// TIA Portal V19 program export: 0 tag tables, 0 data types, 19 data blocks, 51 code blocks (in call order from the OBs), 28 instance data blocks

DATA_BLOCK "A03_DEBUG"   // DB165
// stored: MemoryReserve 100
   VAR
      Force_Sinamics_Infeed_ON : Bool;
      Force_Sinamics_Drives_CtrlSafe : Bool;
      Forse_Contactors_CtrlSafe : Bool;
      LsStratoDepositato : Bool;
      CIn_Manager_DEBUG : Struct
         PareggiatoreTesta : Struct
            Ax : "Positioning_EPOS_Machine_COut";
         END_STRUCT;
         PareggiatoreCoda : Struct
            Ax : "Positioning_EPOS_Machine_COut";
         END_STRUCT;
         Spalle : Struct
            Testa : Struct
               Ax : "Positioning_DOL_Machine_COut";
            END_STRUCT;
            Coda : Struct
               Ax : "Positioning_DOL_Machine_COut";
            END_STRUCT;
         END_STRUCT;
         Spintore : Struct
            Vrt : "ValveMachine_COut";
            Orz : "ValveMachine_COut";
         END_STRUCT;
         TraslazioneStrato : Struct
            Ax_Testa : "Positioning_EPOS_Machine_COut";
            Ax_Coda : "Positioning_EPOS_Machine_COut";
            Manip_Sostegno : "ValveMachine_COut";
            Manip_Pareggiatore : "ValveMachine_COut";
            SostegnoVrt : "ValveMachine_COut";
         END_STRUCT;
         Sollevamento : Struct
            Ax_Testa : "Positioning_DOL_Machine_COut";
            Ax_Coda : "Positioning_DOL_Machine_COut";
         END_STRUCT;
         Sostegno : Struct
            Testa : Struct
               Ax : "Positioning_DOL_Machine_COut";
               Paletto : Struct
                  CtrlSafe : Bool;
                  Standstill : Bool;
                  Rest_CheckNext : Bool;
                  Work_CheckNext : Bool;
                  Pos : Int;
                  RestPosition : Bool;
               END_STRUCT;
            END_STRUCT;
            Coda : Struct
               Ax : "Positioning_DOL_Machine_COut";
               Paletto : Struct
                  CtrlSafe : Bool;
                  Standstill : Bool;
                  Rest_CheckNext : Bool;
                  Work_CheckNext : Bool;
                  Pos : Int;
                  RestPosition : Bool;
               END_STRUCT;
            END_STRUCT;
         END_STRUCT;
         Navetta : Struct
            ReadyToRecive : Bool;
            OutOfWorkspace : Bool;
            InPosizioneDiDeposito : Bool;
            RequestDeposito : Bool;
         END_STRUCT;
         RegolazBord : Struct
            CassettaOP : Real := 65.0;
            LineSetupExe : Bool;
         END_STRUCT;
      END_STRUCT;
      CIn_Manager04_Debug : Struct
         Navetta : Struct
            Testa : Struct
               Ax : "Positioning_DOL_Machine_COut";
               PalettiEsterni : "ValveMachine_COut";
               PalettiInterni : "ValveMachine_COut";
            END_STRUCT;
            Coda : Struct
               Ax : "Positioning_DOL_Machine_COut";
               PalettiEsterni : "ValveMachine_COut";
               PalettiInterni : "ValveMachine_COut";
            END_STRUCT;
            Cumulativo : Struct
               PalettiEsterni : "ValveMachine_COut";
               PalettiInterni : "ValveMachine_COut";
            END_STRUCT;
         END_STRUCT;
         Sollevamento : Struct
            ReadyToDrop : Bool;   // In posizione di deposito e pacco completato
         END_STRUCT;
         Antiribaltamento : Struct
            Work : Bool;
            Rest : Bool;
         END_STRUCT;
      END_STRUCT;
   END_VAR
   VAR RETAIN
      HU_Test : Struct
         Enable : Bool;
         EnableDrive : Bool;
         "Req_Par-Bloccaggio" : Bool;
         "Req_Par-Paregg" : Bool;
         Ctrl_Safe : Bool;
      END_STRUCT;
   END_VAR
   VAR
      test_bitA : Bool;
      test_bitB : Bool;
   END_VAR
   VAR RETAIN
      A0301_Manager : Struct
         BeamCode : Bool;   // 0=Solo Part / 1 = Accoppiamento Part
         "Case" : Int;
         "P1-P3_Init" : Bool;
         "P1-P2_Init" : Bool;
         TrasportoStart : Bool;
         PTrk_Pos1_Write : Bool;
      END_STRUCT;
      A0302_Manager : Struct
         BeamCode : Bool;   // 0=Solo Part / 1 = Accoppiamento Part
         JMP : Bool := TRUE;
         A0303_ReadyToRecive : Bool;
         PareggiaRead : Bool;
         AttrezzamentoBordatrice : Bool;
         BTrk_EXIT_Clear : Bool;
      END_STRUCT;
   END_VAR
   VAR
      A301_PTrk : "PTrk_Item";
   END_VAR
BEGIN
   A301_PTrk.O_ID := 1;
   A301_PTrk.C_ID := 0;
   A301_PTrk.Quality := 0;
   A301_PTrk.Beam_Code := 1;
   A301_PTrk.PLen_Meas := 2700.0;
   A301_PTrk.W_A := 140.0;
   A301_PTrk.H_B := 4.5;
   A301_PTrk.ShiftDone := FALSE;
END_DATA_BLOCK

DATA_BLOCK "PrjConfig_A03"   // DB82
// stored: MemoryReserve 100
   VAR
      Area03_Main : "AreaConfig";
   END_VAR
   VAR RETAIN
      A0301 : Struct
         Fermi_P1 : Struct
            Fermi : Array[1..6] of "ValveMachine_Config";
            Sfalsatore : "ValveMachine_Config";
            DelayMissingCondition : Time := T#3S;
         END_STRUCT;
         Fermi_P2 : Struct
            Fermi : Array[1..6] of "ValveMachine_Config";
            Sollevatori : Array[1..6] of "ValveMachine_Config";
            DelayMissingCondition : Time := T#3S;
         END_STRUCT;
         Fermi_P3 : Struct
            Fermi : Array[1..6] of "ValveMachine_Config";
            DelayMissingCondition : Time := T#3S;
         END_STRUCT;
         Fermi_P4 : Struct
            Fermi : Array[1..6] of "ValveMachine_Config";
            DelayMissingCondition : Time := T#3S;
         END_STRUCT;
         Trasporto { S7_SetPoint := 'True'} : "SpeedMachine_Config";
         Ribaltatore : Struct
            Ax : "Positioning_EPOS_Machine_Config_NEW";
            Solleva_Rib : Array[1..6] of "ValveMachine_Config";
         END_STRUCT;
         SpintoreLaterale : Struct
            Vrt_1 : "ValveMachine_Config";
            Orz_1 : "ValveMachine_Config";
            Vrt_2 : "ValveMachine_Config";
            Orz_2 : "ValveMachine_Config";
            Sollevatori : Array[1..7] of "ValveMachine_Config";
            QuotaIngombro_SpinLat2 : Real := 2680.0;
            QuotaIngombro_SpinLat1 { ExternalWritable := 'False'} : Real := 4777.0;
            DelayMissingCondition : Time := T#500MS;
         END_STRUCT;
      END_STRUCT;
      A0302 : Struct
         Spintore : Struct
            Ax : "Positioning_EPOS_Machine_Config_NEW";
            Vrt : "ValveMachine_Config";
            Orz : "ValveMachine_Config";
            SpintoreLat : Struct
               QuotaIngombro_SpinLat2 : Real := 2680.0;
               QuotaIngombro_SpinLat1 : Real := 4777.0;
            END_STRUCT;
            Bordatrice : Struct
               QuotaIngresso : Real := 801.0;
            END_STRUCT;
            DelayMissingCondition : Time := T#0MS;
         END_STRUCT;
         Bordatrice : Struct
            Ax : "Positioning_EPOS_Machine_Config_NEW";
            Measure : Struct
               K1_CarroPost : LReal := 674.0;   // K1: Misura tra carro di coda e sensore applicato per controllo ingombro pezzo con carro giù
               K2_BancoIngresso : LReal := 3560.0;   // K2: Misura interasse tra lo 0 al centro del banco e la FTC all'uscita della Bordatrice
            END_STRUCT;
         END_STRUCT;
         Regolaz_Bordatrice : Struct
            Formato : Struct
               Ax_D : Array[1..1] of "Positioning_DOL_Machine_Config";
               Ax_M : Array[1..10] of "Positioning_MOL_Machine_Config";
               M1_1 : "Positioning_DOL_Machine_Config";
               M1_2 : "Positioning_DOL_Machine_Config";
               M1_3 : "Positioning_MOL_Machine_Config";
               M1_4 : "Positioning_MOL_Machine_Config";
            END_STRUCT;
         END_STRUCT;
         Rulliera : Struct
            Ax : "SpeedMachine_Config";
         END_STRUCT;
         Centratori : Struct
            Centraggio : Array[1..3] of "ValveMachine_Config";
            Sollevamento : Array[1..3] of "ValveMachine_Config";
            DelayMissingCondition : Time := T#500MS;
            WorkWindows : Struct   // Finestre di disattivazione Centratore 1 e 3 in funzione dei Carri
               Coda : Struct
                  Min : LReal := 300.0;
                  Max : LReal := 1378.0;
               END_STRUCT;
               Testa : Struct
                  Min : LReal := 433.0;
                  Max : LReal := 970.0;
               END_STRUCT;
            END_STRUCT;
         END_STRUCT;
         PareggiatoreCoda : Struct
            Ax : "Positioning_DOL_Machine_Config";
            Bloccaggio : "ValveMachine_Config";
            BattutaVerticale : "ValveMachine_Config";
            PareggiatoreLong : "ValveMachine_Config";
            PosPareggiatore : Struct
               QuotaMin_Work : LReal := 82.0;
               QuotaMax_Work { S7_SetPoint := 'True'} : LReal := 91.0;
            END_STRUCT;
            MinDistanzaConSpalla { S7_SetPoint := 'True'} : LReal := 85.7;
            DelayMissingCondition : Time := T#200MS;
         END_STRUCT;
         PareggiatoreTesta : Struct
            Ax : "Positioning_DOL_Machine_Config";
            Bloccaggio : "ValveMachine_Config";
            Sollevamento : "ValveMachine_Config";
            Centraggio : "ValveMachine_Config";
            MinDistanzaConSpalla : LReal := 5.0;
            DelayMissingCondition : Time := T#200MS;
         END_STRUCT;
         Manipolatore : Struct
            Testa : Struct
               Ax : "Positioning_EPOS_Machine_Config_NEW";
               Sollevatore : "ValveMachine_Config";
               Magnete : "ValveMachine_Config";
            END_STRUCT;
            Coda : Struct
               Ax : "Positioning_EPOS_Machine_Config_NEW";
               Sollevatore : "ValveMachine_Config";
               Magnete : "ValveMachine_Config";
            END_STRUCT;
            DelayMissingCondition : Time := T#200MS;
         END_STRUCT;
      END_STRUCT;
   END_VAR
BEGIN
   Area03_Main.TimeOutStopImmediate := T#1S_500MS;
   Area03_Main.TimeOutStopInPhase := T#10S;
   Area03_Main.TimeOutStopProgrammed := T#5M;
   Area03_Main.TimeOutResetAlarms := T#1S;
   A0301.Fermi_P1.Fermi[1..6].DelayPressureRunningTimeout := T#3S;
   A0301.Fermi_P1.Fermi[1..6].DelayMissingCondition := T#3S;
   A0301.Fermi_P1.Fermi[1..6].Rest_LsQty := 1;
   A0301.Fermi_P1.Fermi[1..6].Work_LsQty := 0;
   A0301.Fermi_P1.Fermi[1..6].Rest_RetainAut := FALSE;
   A0301.Fermi_P1.Fermi[1..6].Work_RetainAut := FALSE;
   A0301.Fermi_P1.Fermi[1..6].V.RestLimSwitchExist := TRUE;
   A0301.Fermi_P1.Fermi[1..6].V.WorkLimSwitchExist := FALSE;
   A0301.Fermi_P1.Fermi[1..6].V.CheckOilInPressure := FALSE;
   A0301.Fermi_P1.Fermi[1..6].V.CutRestWhenIsAtRest := TRUE;
   A0301.Fermi_P1.Fermi[1..6].V.CutWorkWhenIsAtWork := FALSE;
   A0301.Fermi_P1.Fermi[1..6].V.RestTime := T#1MS;
   A0301.Fermi_P1.Fermi[1..6].V.WorkTime := T#100MS;
   A0301.Fermi_P1.Fermi[1..6].V.RestTimeOut := T#4S;
   A0301.Fermi_P1.Fermi[1..6].V.WorkTimeOut := T#4S;
   A0301.Fermi_P1.Sfalsatore.DelayPressureRunningTimeout := T#3S;
   A0301.Fermi_P1.Sfalsatore.DelayMissingCondition := T#3S;
   A0301.Fermi_P1.Sfalsatore.Rest_LsQty := 1;
   A0301.Fermi_P1.Sfalsatore.Work_LsQty := 1;
   A0301.Fermi_P1.Sfalsatore.Rest_RetainAut := FALSE;
   A0301.Fermi_P1.Sfalsatore.Work_RetainAut := FALSE;
   A0301.Fermi_P1.Sfalsatore.V.RestLimSwitchExist := TRUE;
   A0301.Fermi_P1.Sfalsatore.V.WorkLimSwitchExist := TRUE;
   A0301.Fermi_P1.Sfalsatore.V.CheckOilInPressure := FALSE;
   A0301.Fermi_P1.Sfalsatore.V.CutRestWhenIsAtRest := FALSE;
   A0301.Fermi_P1.Sfalsatore.V.CutWorkWhenIsAtWork := TRUE;
   A0301.Fermi_P1.Sfalsatore.V.RestTime := T#1S;
   A0301.Fermi_P1.Sfalsatore.V.WorkTime := T#300MS;
   A0301.Fermi_P1.Sfalsatore.V.RestTimeOut := T#1H;
   A0301.Fermi_P1.Sfalsatore.V.WorkTimeOut := T#1H;
   A0301.Fermi_P2.Fermi[1..6].DelayPressureRunningTimeout := T#3S;
   A0301.Fermi_P2.Fermi[1..6].DelayMissingCondition := T#3S;
   A0301.Fermi_P2.Fermi[1..6].Rest_LsQty := 1;
   A0301.Fermi_P2.Fermi[1..6].Work_LsQty := 0;
   A0301.Fermi_P2.Fermi[1..6].Rest_RetainAut := FALSE;
   A0301.Fermi_P2.Fermi[1..6].Work_RetainAut := FALSE;
   A0301.Fermi_P2.Fermi[1..6].V.RestLimSwitchExist := TRUE;
   A0301.Fermi_P2.Fermi[1..6].V.WorkLimSwitchExist := FALSE;
   A0301.Fermi_P2.Fermi[1..6].V.CheckOilInPressure := FALSE;
   A0301.Fermi_P2.Fermi[1..6].V.CutRestWhenIsAtRest := TRUE;
   A0301.Fermi_P2.Fermi[1..6].V.CutWorkWhenIsAtWork := FALSE;
   A0301.Fermi_P2.Fermi[1..6].V.RestTime := T#1MS;
   A0301.Fermi_P2.Fermi[1..6].V.WorkTime := T#100MS;
   A0301.Fermi_P2.Fermi[1..6].V.RestTimeOut := T#4S;
   A0301.Fermi_P2.Fermi[1..6].V.WorkTimeOut := T#4S;
   A0301.Fermi_P2.Sollevatori[1..6].DelayPressureRunningTimeout := T#3S;
   A0301.Fermi_P2.Sollevatori[1..6].DelayMissingCondition := T#3S;
   A0301.Fermi_P2.Sollevatori[1..6].Rest_LsQty := 1;
   A0301.Fermi_P2.Sollevatori[1..6].Work_LsQty := 0;
   A0301.Fermi_P2.Sollevatori[1..6].Rest_RetainAut := FALSE;
   A0301.Fermi_P2.Sollevatori[1..6].Work_RetainAut := FALSE;
   A0301.Fermi_P2.Sollevatori[1..6].V.RestLimSwitchExist := TRUE;
   A0301.Fermi_P2.Sollevatori[1..6].V.WorkLimSwitchExist := FALSE;
   A0301.Fermi_P2.Sollevatori[1..6].V.CheckOilInPressure := FALSE;
   A0301.Fermi_P2.Sollevatori[1..6].V.CutRestWhenIsAtRest := TRUE;
   A0301.Fermi_P2.Sollevatori[1..6].V.CutWorkWhenIsAtWork := FALSE;
   A0301.Fermi_P2.Sollevatori[1..6].V.RestTime := T#1MS;
   A0301.Fermi_P2.Sollevatori[1..6].V.WorkTime := T#100MS;
   A0301.Fermi_P2.Sollevatori[1..6].V.RestTimeOut := T#4S;
   A0301.Fermi_P2.Sollevatori[1..6].V.WorkTimeOut := T#4S;
   A0301.Fermi_P3.Fermi[1..6].DelayPressureRunningTimeout := T#3S;
   A0301.Fermi_P3.Fermi[1..6].DelayMissingCondition := T#3S;
   A0301.Fermi_P3.Fermi[1..6].Rest_LsQty := 1;
   A0301.Fermi_P3.Fermi[1..6].Work_LsQty := 0;
   A0301.Fermi_P3.Fermi[1..6].Rest_RetainAut := FALSE;
   A0301.Fermi_P3.Fermi[1..6].Work_RetainAut := FALSE;
   A0301.Fermi_P3.Fermi[1..6].V.RestLimSwitchExist := TRUE;
   A0301.Fermi_P3.Fermi[1..6].V.WorkLimSwitchExist := FALSE;
   A0301.Fermi_P3.Fermi[1..6].V.CheckOilInPressure := FALSE;
   A0301.Fermi_P3.Fermi[1..6].V.CutRestWhenIsAtRest := TRUE;
   A0301.Fermi_P3.Fermi[1..6].V.CutWorkWhenIsAtWork := FALSE;
   A0301.Fermi_P3.Fermi[1..6].V.RestTime := T#1MS;
   A0301.Fermi_P3.Fermi[1..6].V.WorkTime := T#100MS;
   A0301.Fermi_P3.Fermi[1..6].V.RestTimeOut := T#4S;
   A0301.Fermi_P3.Fermi[1..6].V.WorkTimeOut := T#4S;
   A0301.Fermi_P4.Fermi[1..6].DelayPressureRunningTimeout := T#3S;
   A0301.Fermi_P4.Fermi[1..6].DelayMissingCondition := T#3S;
   A0301.Fermi_P4.Fermi[1..6].Rest_LsQty := 1;
   A0301.Fermi_P4.Fermi[1..6].Work_LsQty := 0;
   A0301.Fermi_P4.Fermi[1..6].Rest_RetainAut := FALSE;
   A0301.Fermi_P4.Fermi[1..6].Work_RetainAut := FALSE;
   A0301.Fermi_P4.Fermi[1..6].V.RestLimSwitchExist := TRUE;
   A0301.Fermi_P4.Fermi[1..6].V.WorkLimSwitchExist := FALSE;
   A0301.Fermi_P4.Fermi[1..6].V.CheckOilInPressure := FALSE;
   A0301.Fermi_P4.Fermi[1..6].V.CutRestWhenIsAtRest := TRUE;
   A0301.Fermi_P4.Fermi[1..6].V.CutWorkWhenIsAtWork := FALSE;
   A0301.Fermi_P4.Fermi[1..6].V.RestTime := T#1MS;
   A0301.Fermi_P4.Fermi[1..6].V.WorkTime := T#300MS;
   A0301.Fermi_P4.Fermi[1..6].V.RestTimeOut := T#4S;
   A0301.Fermi_P4.Fermi[1..6].V.WorkTimeOut := T#4S;
   A0301.Trasporto.SLS_VEL := 5000.0;
   A0301.Trasporto.DelayMissingCondition := T#3S;
   A0301.Trasporto.Ax.SINA_Drive.ReferenceVelocity := 2200.0;
   A0301.Trasporto.Ax.SINA_Drive.InvertDirection := FALSE;
   A0301.Trasporto.Ax.MinAccTime := 0.1;
   A0301.Trasporto.Ax.MinDecTime := 0.1;
   A0301.Trasporto.Ax.LeadScrewPitchVal := 359.8;
   A0301.Trasporto.Ax.MotorRevolution := 20.0;
   A0301.Trasporto.Ax.LoadRevolution := 1.0;
   A0301.Trasporto.Ax.PowerOffDelay := T#1S_500MS;
   A0301.Trasporto.Ax.StandstillVelocity := 50.0;
   A0301.Trasporto.Ax.StandstillDelay := T#100MS;
   A0301.Trasporto.Fan.Presence := FALSE;
   A0301.Trasporto.Fan.DelayOff := T#0MS;
   A0301.Trasporto.Brake_Presence := FALSE;
   A0301.Ribaltatore.Ax.SLS_Vel := 3000.0;
   A0301.Ribaltatore.Ax.DelayMissingCondition := T#100MS;
   A0301.Ribaltatore.Ax.Ax.Encoder_Inc_AutoReloadPosition := FALSE;
   A0301.Ribaltatore.Ax.Ax.Encoder_is_Absolute := TRUE;
   A0301.Ribaltatore.Ax.Ax.LeadScrewPitchVal := 9.0000015;
   A0301.Ribaltatore.Ax.Ax.MotorRevolution := 23.33;
   A0301.Ribaltatore.Ax.Ax.LoadRevolution := 1.0;
   A0301.Ribaltatore.Ax.Ax.PowerOffDelay := T#100MS;
   A0301.Ribaltatore.Ax.Ax.MaxRPM_S120_P2000 := 3000.0;
   A0301.Ribaltatore.Ax.Ax.MaxVel_S120_P2571 := 6000.0;
   A0301.Ribaltatore.Ax.Ax.MaxAcc_S120_P2572 := 50.0;
   A0301.Ribaltatore.Ax.Ax.MaxDec_S120_P2573 := 50.0;
   A0301.Ribaltatore.Ax.Ax.Modulo_S120_P2566 := 0.0;
   A0301.Ribaltatore.Ax.Ax.SwLimMinus_S120_P2580 := 0.25;
   A0301.Ribaltatore.Ax.Ax.SwLimPlus_S120_P2581 := 125.0;
   A0301.Ribaltatore.Ax.Fan.Presence := FALSE;
   A0301.Ribaltatore.Ax.Fan.DelayOff := T#0MS;
   A0301.Ribaltatore.Ax.Brake_Presence := FALSE;
   A0301.Ribaltatore.Solleva_Rib[1..6].DelayPressureRunningTimeout := T#3S;
   A0301.Ribaltatore.Solleva_Rib[1..6].DelayMissingCondition := T#3S;
   A0301.Ribaltatore.Solleva_Rib[1..6].Rest_LsQty := 1;
   A0301.Ribaltatore.Solleva_Rib[1..6].Work_LsQty := 1;
   A0301.Ribaltatore.Solleva_Rib[1..6].Rest_RetainAut := FALSE;
   A0301.Ribaltatore.Solleva_Rib[1..6].Work_RetainAut := FALSE;
   A0301.Ribaltatore.Solleva_Rib[1..6].V.RestLimSwitchExist := TRUE;
   A0301.Ribaltatore.Solleva_Rib[1..6].V.WorkLimSwitchExist := TRUE;
   A0301.Ribaltatore.Solleva_Rib[1..6].V.CheckOilInPressure := FALSE;
   A0301.Ribaltatore.Solleva_Rib[1..6].V.CutRestWhenIsAtRest := FALSE;
   A0301.Ribaltatore.Solleva_Rib[1..6].V.CutWorkWhenIsAtWork := FALSE;
   A0301.Ribaltatore.Solleva_Rib[1..6].V.RestTime := T#1MS;
   A0301.Ribaltatore.Solleva_Rib[1..6].V.WorkTime := T#200MS;
   A0301.Ribaltatore.Solleva_Rib[1..6].V.RestTimeOut := T#5S;
   A0301.Ribaltatore.Solleva_Rib[1..6].V.WorkTimeOut := T#5S;
   A0301.SpintoreLaterale.Vrt_1.DelayPressureRunningTimeout := T#3S;
   A0301.SpintoreLaterale.Vrt_1.DelayMissingCondition := T#3S;
   A0301.SpintoreLaterale.Vrt_1.Rest_LsQty := 1;
   A0301.SpintoreLaterale.Vrt_1.Work_LsQty := 0;
   A0301.SpintoreLaterale.Vrt_1.Rest_RetainAut := FALSE;
   A0301.SpintoreLaterale.Vrt_1.Work_RetainAut := FALSE;
   A0301.SpintoreLaterale.Vrt_1.V.RestLimSwitchExist := TRUE;
   A0301.SpintoreLaterale.Vrt_1.V.WorkLimSwitchExist := FALSE;
   A0301.SpintoreLaterale.Vrt_1.V.CheckOilInPressure := FALSE;
   A0301.SpintoreLaterale.Vrt_1.V.CutRestWhenIsAtRest := TRUE;
   A0301.SpintoreLaterale.Vrt_1.V.CutWorkWhenIsAtWork := FALSE;
   A0301.SpintoreLaterale.Vrt_1.V.RestTime := T#1MS;
   A0301.SpintoreLaterale.Vrt_1.V.WorkTime := T#300MS;
   A0301.SpintoreLaterale.Vrt_1.V.RestTimeOut := T#5S;
   A0301.SpintoreLaterale.Vrt_1.V.WorkTimeOut := T#5S;
   A0301.SpintoreLaterale.Orz_1.DelayPressureRunningTimeout := T#3S;
   A0301.SpintoreLaterale.Orz_1.DelayMissingCondition := T#3S;
   A0301.SpintoreLaterale.Orz_1.Rest_LsQty := 1;
   A0301.SpintoreLaterale.Orz_1.Work_LsQty := 0;
   A0301.SpintoreLaterale.Orz_1.Rest_RetainAut := FALSE;
   A0301.SpintoreLaterale.Orz_1.Work_RetainAut := FALSE;
   A0301.SpintoreLaterale.Orz_1.V.RestLimSwitchExist := TRUE;
   A0301.SpintoreLaterale.Orz_1.V.WorkLimSwitchExist := FALSE;
   A0301.SpintoreLaterale.Orz_1.V.CheckOilInPressure := FALSE;
   A0301.SpintoreLaterale.Orz_1.V.CutRestWhenIsAtRest := FALSE;
   A0301.SpintoreLaterale.Orz_1.V.CutWorkWhenIsAtWork := FALSE;
   A0301.SpintoreLaterale.Orz_1.V.RestTime := T#1MS;
   A0301.SpintoreLaterale.Orz_1.V.WorkTime := T#300MS;
   A0301.SpintoreLaterale.Orz_1.V.RestTimeOut := T#5S;
   A0301.SpintoreLaterale.Orz_1.V.WorkTimeOut := T#5S;
   A0301.SpintoreLaterale.Vrt_2.DelayPressureRunningTimeout := T#3S;
   A0301.SpintoreLaterale.Vrt_2.DelayMissingCondition := T#3S;
   A0301.SpintoreLaterale.Vrt_2.Rest_LsQty := 1;
   A0301.SpintoreLaterale.Vrt_2.Work_LsQty := 0;
   A0301.SpintoreLaterale.Vrt_2.Rest_RetainAut := FALSE;
   A0301.SpintoreLaterale.Vrt_2.Work_RetainAut := FALSE;
   A0301.SpintoreLaterale.Vrt_2.V.RestLimSwitchExist := TRUE;
   A0301.SpintoreLaterale.Vrt_2.V.WorkLimSwitchExist := FALSE;
   A0301.SpintoreLaterale.Vrt_2.V.CheckOilInPressure := FALSE;
   A0301.SpintoreLaterale.Vrt_2.V.CutRestWhenIsAtRest := TRUE;
   A0301.SpintoreLaterale.Vrt_2.V.CutWorkWhenIsAtWork := FALSE;
   A0301.SpintoreLaterale.Vrt_2.V.RestTime := T#1MS;
   A0301.SpintoreLaterale.Vrt_2.V.WorkTime := T#300MS;
   A0301.SpintoreLaterale.Vrt_2.V.RestTimeOut := T#5S;
   A0301.SpintoreLaterale.Vrt_2.V.WorkTimeOut := T#5S;
   A0301.SpintoreLaterale.Orz_2.DelayPressureRunningTimeout := T#3S;
   A0301.SpintoreLaterale.Orz_2.DelayMissingCondition := T#3S;
   A0301.SpintoreLaterale.Orz_2.Rest_LsQty := 1;
   A0301.SpintoreLaterale.Orz_2.Work_LsQty := 0;
   A0301.SpintoreLaterale.Orz_2.Rest_RetainAut := FALSE;
   A0301.SpintoreLaterale.Orz_2.Work_RetainAut := FALSE;
   A0301.SpintoreLaterale.Orz_2.V.RestLimSwitchExist := TRUE;
   A0301.SpintoreLaterale.Orz_2.V.WorkLimSwitchExist := FALSE;
   A0301.SpintoreLaterale.Orz_2.V.CheckOilInPressure := FALSE;
   A0301.SpintoreLaterale.Orz_2.V.CutRestWhenIsAtRest := FALSE;
   A0301.SpintoreLaterale.Orz_2.V.CutWorkWhenIsAtWork := FALSE;
   A0301.SpintoreLaterale.Orz_2.V.RestTime := T#1MS;
   A0301.SpintoreLaterale.Orz_2.V.WorkTime := T#300MS;
   A0301.SpintoreLaterale.Orz_2.V.RestTimeOut := T#5S;
   A0301.SpintoreLaterale.Orz_2.V.WorkTimeOut := T#5S;
   A0301.SpintoreLaterale.Sollevatori[1..7].DelayPressureRunningTimeout := T#3S;
   A0301.SpintoreLaterale.Sollevatori[1..7].DelayMissingCondition := T#3S;
   A0301.SpintoreLaterale.Sollevatori[1..7].Rest_LsQty := 1;
   A0301.SpintoreLaterale.Sollevatori[1..7].Work_LsQty := 0;
   A0301.SpintoreLaterale.Sollevatori[1..7].Rest_RetainAut := FALSE;
   A0301.SpintoreLaterale.Sollevatori[1..7].Work_RetainAut := FALSE;
   A0301.SpintoreLaterale.Sollevatori[1..7].V.RestLimSwitchExist := TRUE;
   A0301.SpintoreLaterale.Sollevatori[1..7].V.WorkLimSwitchExist := FALSE;
   A0301.SpintoreLaterale.Sollevatori[1..7].V.CheckOilInPressure := FALSE;
   A0301.SpintoreLaterale.Sollevatori[1..7].V.CutRestWhenIsAtRest := TRUE;
   A0301.SpintoreLaterale.Sollevatori[1..7].V.CutWorkWhenIsAtWork := TRUE;
   A0301.SpintoreLaterale.Sollevatori[1..7].V.RestTime := T#1S;
   A0301.SpintoreLaterale.Sollevatori[1..7].V.WorkTime := T#500MS;
   A0301.SpintoreLaterale.Sollevatori[1..7].V.RestTimeOut := T#4S;
   A0301.SpintoreLaterale.Sollevatori[1..7].V.WorkTimeOut := T#4S;
   A0302.Spintore.Ax.SLS_Vel := 3000.0;
   A0302.Spintore.Ax.DelayMissingCondition := T#1S;
   A0302.Spintore.Ax.Ax.Encoder_Inc_AutoReloadPosition := FALSE;
   A0302.Spintore.Ax.Ax.Encoder_is_Absolute := TRUE;
   A0302.Spintore.Ax.Ax.LeadScrewPitchVal := 287.989799;
   A0302.Spintore.Ax.Ax.MotorRevolution := 10.0;
   A0302.Spintore.Ax.Ax.LoadRevolution := 1.0;
   A0302.Spintore.Ax.Ax.PowerOffDelay := T#1S;
   A0302.Spintore.Ax.Ax.MaxRPM_S120_P2000 := 3000.0;
   A0302.Spintore.Ax.Ax.MaxVel_S120_P2571 := 86396.0;
   A0302.Spintore.Ax.Ax.MaxAcc_S120_P2572 := 5000.0;
   A0302.Spintore.Ax.Ax.MaxDec_S120_P2573 := 5000.0;
   A0302.Spintore.Ax.Ax.Modulo_S120_P2566 := 0.0;
   A0302.Spintore.Ax.Ax.SwLimMinus_S120_P2580 := 0.5;
   A0302.Spintore.Ax.Ax.SwLimPlus_S120_P2581 := 5370.0;
   A0302.Spintore.Ax.Fan.Presence := FALSE;
   A0302.Spintore.Ax.Fan.DelayOff := T#0MS;
   A0302.Spintore.Ax.Brake_Presence := FALSE;
   A0302.Spintore.Vrt.DelayPressureRunningTimeout := T#3S;
   A0302.Spintore.Vrt.DelayMissingCondition := T#3S;
   A0302.Spintore.Vrt.Rest_LsQty := 1;
   A0302.Spintore.Vrt.Work_LsQty := 1;
   A0302.Spintore.Vrt.Rest_RetainAut := FALSE;
   A0302.Spintore.Vrt.Work_RetainAut := FALSE;
   A0302.Spintore.Vrt.V.RestLimSwitchExist := TRUE;
   A0302.Spintore.Vrt.V.WorkLimSwitchExist := TRUE;
   A0302.Spintore.Vrt.V.CheckOilInPressure := FALSE;
   A0302.Spintore.Vrt.V.CutRestWhenIsAtRest := TRUE;
   A0302.Spintore.Vrt.V.CutWorkWhenIsAtWork := FALSE;
   A0302.Spintore.Vrt.V.RestTime := T#10MS;
   A0302.Spintore.Vrt.V.WorkTime := T#100MS;
   A0302.Spintore.Vrt.V.RestTimeOut := T#4S;
   A0302.Spintore.Vrt.V.WorkTimeOut := T#4S;
   A0302.Spintore.Orz.DelayPressureRunningTimeout := T#3S;
   A0302.Spintore.Orz.DelayMissingCondition := T#3S;
   A0302.Spintore.Orz.Rest_LsQty := 1;
   A0302.Spintore.Orz.Work_LsQty := 0;
   A0302.Spintore.Orz.Rest_RetainAut := FALSE;
   A0302.Spintore.Orz.Work_RetainAut := FALSE;
   A0302.Spintore.Orz.V.RestLimSwitchExist := TRUE;
   A0302.Spintore.Orz.V.WorkLimSwitchExist := FALSE;
   A0302.Spintore.Orz.V.CheckOilInPressure := FALSE;
   A0302.Spintore.Orz.V.CutRestWhenIsAtRest := TRUE;
   A0302.Spintore.Orz.V.CutWorkWhenIsAtWork := FALSE;
   A0302.Spintore.Orz.V.RestTime := T#10MS;
   A0302.Spintore.Orz.V.WorkTime := T#100MS;
   A0302.Spintore.Orz.V.RestTimeOut := T#4S;
   A0302.Spintore.Orz.V.WorkTimeOut := T#4S;
   A0302.Bordatrice.Ax.SLS_Vel := 3000.0;
   A0302.Bordatrice.Ax.DelayMissingCondition := T#200MS;
   A0302.Bordatrice.Ax.Ax.Encoder_Inc_AutoReloadPosition := TRUE;
   A0302.Bordatrice.Ax.Ax.Encoder_is_Absolute := FALSE;
   A0302.Bordatrice.Ax.Ax.LeadScrewPitchVal := 486.946;
   A0302.Bordatrice.Ax.Ax.MotorRevolution := 12.4;
   A0302.Bordatrice.Ax.Ax.LoadRevolution := 1.0;
   A0302.Bordatrice.Ax.Ax.PowerOffDelay := T#500MS;
   A0302.Bordatrice.Ax.Ax.MaxRPM_S120_P2000 := 3000.0;
   A0302.Bordatrice.Ax.Ax.MaxVel_S120_P2571 := 60000.0;
   A0302.Bordatrice.Ax.Ax.MaxAcc_S120_P2572 := 4000.0;
   A0302.Bordatrice.Ax.Ax.MaxDec_S120_P2573 := 4000.0;
   A0302.Bordatrice.Ax.Ax.Modulo_S120_P2566 := 1000000000.0;
   A0302.Bordatrice.Ax.Ax.SwLimMinus_S120_P2580 := 0.0;
   A0302.Bordatrice.Ax.Ax.SwLimPlus_S120_P2581 := 0.0;
   A0302.Bordatrice.Ax.Fan.Presence := FALSE;
   A0302.Bordatrice.Ax.Fan.DelayOff := T#0MS;
   A0302.Bordatrice.Ax.Brake_Presence := FALSE;
   A0302.Regolaz_Bordatrice.Formato.Ax_D[1].DelayMissingCondition := T#3S;
   A0302.Regolaz_Bordatrice.Formato.Ax_D[1].CyclicOBTime_ms := 10.0;
   A0302.Regolaz_Bordatrice.Formato.Ax_D[1].Ax.limitMinus := 59.0;
   A0302.Regolaz_Bordatrice.Formato.Ax_D[1].Ax.limitPlus := 215.0;
   A0302.Regolaz_Bordatrice.Formato.Ax_D[1].Ax.Backlash := 0.4;
   A0302.Regolaz_Bordatrice.Formato.Ax_D[1].Ax.BacklashActivation := TRUE;
   A0302.Regolaz_Bordatrice.Formato.Ax_D[1].Ax.ToleranceWindow := 0.0;
   A0302.Regolaz_Bordatrice.Formato.Ax_D[1].Ax.ToleranceWindowDelay := T#100MS;
   A0302.Regolaz_Bordatrice.Formato.Ax_D[1].Ax.PreCutOff := 0.03;
   A0302.Regolaz_Bordatrice.Formato.Ax_D[1].Ax.PreEndLowSpeed := 0.0;
   A0302.Regolaz_Bordatrice.Formato.Ax_D[1].Ax.PreEndMedSpeed := 0.0;
   A0302.Regolaz_Bordatrice.Formato.Ax_D[1].Ax.ChangeDirectionDelay := T#0MS;
   A0302.Regolaz_Bordatrice.Formato.Ax_D[1].Ax.StandstillVelocity := 0.5;
   A0302.Regolaz_Bordatrice.Formato.Ax_D[1].Ax.StandStillDelay := T#100MS;
   A0302.Regolaz_Bordatrice.Formato.Ax_D[1].Ax.HomingDirection := FALSE;
   A0302.Regolaz_Bordatrice.Formato.Ax_D[1].Ax.RecallTime := 0.0;
   A0302.Regolaz_Bordatrice.Formato.Ax_D[1].Ax.VelocityFilter_T := 10.0;
   A0302.Regolaz_Bordatrice.Formato.Ax_D[1].Ax.VelocityMeasUnit := 2;
   A0302.Regolaz_Bordatrice.Formato.Ax_D[1].Ax.PosFbkDisabled := FALSE;
   A0302.Regolaz_Bordatrice.Formato.Ax_D[1].Ax.FbkCtrlDisabled := TRUE;
   A0302.Regolaz_Bordatrice.Formato.Ax_D[1].Ax_UM2."m" := -1.0;
   A0302.Regolaz_Bordatrice.Formato.Ax_D[1].Ax_UM2.q := 320.5;
   A0302.Regolaz_Bordatrice.Formato.Ax_D[1].S120.SpeedMotor.ReferenceVelocity := 2200.0;
   A0302.Regolaz_Bordatrice.Formato.Ax_D[1].S120.SpeedMotor.InvertDirection := FALSE;
   A0302.Regolaz_Bordatrice.Formato.Ax_D[1].S120.PowerOffDelay := T#1S_500MS;
   A0302.Regolaz_Bordatrice.Formato.Ax_D[1].S120.StandstillVelocity := 20.0;
   A0302.Regolaz_Bordatrice.Formato.Ax_D[1].S120.AccTime := 0.5;
   A0302.Regolaz_Bordatrice.Formato.Ax_D[1].S120.DecTime := 0.5;
   A0302.Regolaz_Bordatrice.Formato.Ax_D[1].Fan.Presence := FALSE;
   A0302.Regolaz_Bordatrice.Formato.Ax_D[1].Fan.DelayOff := T#10M;
   A0302.Regolaz_Bordatrice.Formato.Ax_D[1].Brake_Presence := FALSE;
   A0302.Regolaz_Bordatrice.Formato.Ax_M[1..10].DelayMissingCondition := T#100MS;
   A0302.Regolaz_Bordatrice.Formato.Ax_M[1..10].CyclicOBTime_ms := 10.0;
   A0302.Regolaz_Bordatrice.Formato.Ax_M[1..10].Ax.limitMinus := 38.0;
   A0302.Regolaz_Bordatrice.Formato.Ax_M[1..10].Ax.limitPlus := 52.0;
   A0302.Regolaz_Bordatrice.Formato.Ax_M[1..10].Ax.Backlash := 0.4;
   A0302.Regolaz_Bordatrice.Formato.Ax_M[1..10].Ax.BacklashActivation := TRUE;
   A0302.Regolaz_Bordatrice.Formato.Ax_M[1..10].Ax.ToleranceWindow := 0.0;
   A0302.Regolaz_Bordatrice.Formato.Ax_M[1..10].Ax.ToleranceWindowDelay := T#100MS;
   A0302.Regolaz_Bordatrice.Formato.Ax_M[1..10].Ax.PreCutOff := 0.03;
   A0302.Regolaz_Bordatrice.Formato.Ax_M[1..10].Ax.PreEndLowSpeed := 0.0;
   A0302.Regolaz_Bordatrice.Formato.Ax_M[1..10].Ax.PreEndMedSpeed := 0.0;
   A0302.Regolaz_Bordatrice.Formato.Ax_M[1..10].Ax.ChangeDirectionDelay := T#0MS;
   A0302.Regolaz_Bordatrice.Formato.Ax_M[1..10].Ax.StandstillVelocity := 0.5;
   A0302.Regolaz_Bordatrice.Formato.Ax_M[1..10].Ax.StandStillDelay := T#100MS;
   A0302.Regolaz_Bordatrice.Formato.Ax_M[1..10].Ax.HomingDirection := FALSE;
   A0302.Regolaz_Bordatrice.Formato.Ax_M[1..10].Ax.RecallTime := 0.0;
   A0302.Regolaz_Bordatrice.Formato.Ax_M[1..10].Ax.VelocityFilter_T := 10.0;
   A0302.Regolaz_Bordatrice.Formato.Ax_M[1..10].Ax.VelocityMeasUnit := 2;
   A0302.Regolaz_Bordatrice.Formato.Ax_M[1..10].Ax.PosFbkDisabled := FALSE;
   A0302.Regolaz_Bordatrice.Formato.Ax_M[1..10].Ax.FbkCtrlDisabled := TRUE;
   A0302.Regolaz_Bordatrice.Formato.Ax_M[1..10].Ax_UM2."m" := 1.0;
   A0302.Regolaz_Bordatrice.Formato.Ax_M[1..5].Ax_UM2.q := 127.0;
   A0302.Regolaz_Bordatrice.Formato.Ax_M[6..10].Ax_UM2.q := 84.8;
   A0302.Regolaz_Bordatrice.Formato.M1_1.DelayMissingCondition := T#3S;
   A0302.Regolaz_Bordatrice.Formato.M1_1.CyclicOBTime_ms := 10.0;
   A0302.Regolaz_Bordatrice.Formato.M1_1.Ax.limitMinus := 0.0;
   A0302.Regolaz_Bordatrice.Formato.M1_1.Ax.limitPlus := 0.0;
   A0302.Regolaz_Bordatrice.Formato.M1_1.Ax.Backlash := 0.0;
   A0302.Regolaz_Bordatrice.Formato.M1_1.Ax.BacklashActivation := FALSE;
   A0302.Regolaz_Bordatrice.Formato.M1_1.Ax.ToleranceWindow := 0.0;
   A0302.Regolaz_Bordatrice.Formato.M1_1.Ax.ToleranceWindowDelay := T#0MS;
   A0302.Regolaz_Bordatrice.Formato.M1_1.Ax.PreCutOff := 0.0;
   A0302.Regolaz_Bordatrice.Formato.M1_1.Ax.PreEndLowSpeed := 0.0;
   A0302.Regolaz_Bordatrice.Formato.M1_1.Ax.PreEndMedSpeed := 0.0;
   A0302.Regolaz_Bordatrice.Formato.M1_1.Ax.ChangeDirectionDelay := T#0MS;
   A0302.Regolaz_Bordatrice.Formato.M1_1.Ax.StandstillVelocity := 0.0;
   A0302.Regolaz_Bordatrice.Formato.M1_1.Ax.StandStillDelay := T#0MS;
   A0302.Regolaz_Bordatrice.Formato.M1_1.Ax.HomingDirection := FALSE;
   A0302.Regolaz_Bordatrice.Formato.M1_1.Ax.RecallTime := 0.0;
   A0302.Regolaz_Bordatrice.Formato.M1_1.Ax.VelocityFilter_T := 10.0;
   A0302.Regolaz_Bordatrice.Formato.M1_1.Ax.VelocityMeasUnit := 0;
   A0302.Regolaz_Bordatrice.Formato.M1_1.Ax.PosFbkDisabled := FALSE;
   A0302.Regolaz_Bordatrice.Formato.M1_1.Ax.FbkCtrlDisabled := FALSE;
   A0302.Regolaz_Bordatrice.Formato.M1_1.Ax_UM2."m" := 1.0;
   A0302.Regolaz_Bordatrice.Formato.M1_1.Ax_UM2.q := 0.0;
   A0302.Regolaz_Bordatrice.Formato.M1_1.S120.SpeedMotor.ReferenceVelocity := 2000.0;
   A0302.Regolaz_Bordatrice.Formato.M1_1.S120.SpeedMotor.InvertDirection := FALSE;
   A0302.Regolaz_Bordatrice.Formato.M1_1.S120.PowerOffDelay := T#1S_500MS;
   A0302.Regolaz_Bordatrice.Formato.M1_1.S120.StandstillVelocity := 0.0;
   A0302.Regolaz_Bordatrice.Formato.M1_1.S120.AccTime := 0.0;
   A0302.Regolaz_Bordatrice.Formato.M1_1.S120.DecTime := 0.0;
   A0302.Regolaz_Bordatrice.Formato.M1_1.Fan.Presence := FALSE;
   A0302.Regolaz_Bordatrice.Formato.M1_1.Fan.DelayOff := T#10M;
   A0302.Regolaz_Bordatrice.Formato.M1_1.Brake_Presence := FALSE;
   A0302.Regolaz_Bordatrice.Formato.M1_2.DelayMissingCondition := T#3S;
   A0302.Regolaz_Bordatrice.Formato.M1_2.CyclicOBTime_ms := 10.0;
   A0302.Regolaz_Bordatrice.Formato.M1_2.Ax.limitMinus := 0.0;
   A0302.Regolaz_Bordatrice.Formato.M1_2.Ax.limitPlus := 0.0;
   A0302.Regolaz_Bordatrice.Formato.M1_2.Ax.Backlash := 0.0;
   A0302.Regolaz_Bordatrice.Formato.M1_2.Ax.BacklashActivation := FALSE;
   A0302.Regolaz_Bordatrice.Formato.M1_2.Ax.ToleranceWindow := 0.0;
   A0302.Regolaz_Bordatrice.Formato.M1_2.Ax.ToleranceWindowDelay := T#0MS;
   A0302.Regolaz_Bordatrice.Formato.M1_2.Ax.PreCutOff := 0.0;
   A0302.Regolaz_Bordatrice.Formato.M1_2.Ax.PreEndLowSpeed := 0.0;
   A0302.Regolaz_Bordatrice.Formato.M1_2.Ax.PreEndMedSpeed := 0.0;
   A0302.Regolaz_Bordatrice.Formato.M1_2.Ax.ChangeDirectionDelay := T#0MS;
   A0302.Regolaz_Bordatrice.Formato.M1_2.Ax.StandstillVelocity := 0.0;
   A0302.Regolaz_Bordatrice.Formato.M1_2.Ax.StandStillDelay := T#0MS;
   A0302.Regolaz_Bordatrice.Formato.M1_2.Ax.HomingDirection := FALSE;
   A0302.Regolaz_Bordatrice.Formato.M1_2.Ax.RecallTime := 0.0;
   A0302.Regolaz_Bordatrice.Formato.M1_2.Ax.VelocityFilter_T := 10.0;
   A0302.Regolaz_Bordatrice.Formato.M1_2.Ax.VelocityMeasUnit := 0;
   A0302.Regolaz_Bordatrice.Formato.M1_2.Ax.PosFbkDisabled := FALSE;
   A0302.Regolaz_Bordatrice.Formato.M1_2.Ax.FbkCtrlDisabled := FALSE;
   A0302.Regolaz_Bordatrice.Formato.M1_2.Ax_UM2."m" := 1.0;
   A0302.Regolaz_Bordatrice.Formato.M1_2.Ax_UM2.q := 0.0;
   A0302.Regolaz_Bordatrice.Formato.M1_2.S120.SpeedMotor.ReferenceVelocity := 2000.0;
   A0302.Regolaz_Bordatrice.Formato.M1_2.S120.SpeedMotor.InvertDirection := FALSE;
   A0302.Regolaz_Bordatrice.Formato.M1_2.S120.PowerOffDelay := T#1S_500MS;
   A0302.Regolaz_Bordatrice.Formato.M1_2.S120.StandstillVelocity := 0.0;
   A0302.Regolaz_Bordatrice.Formato.M1_2.S120.AccTime := 0.0;
   A0302.Regolaz_Bordatrice.Formato.M1_2.S120.DecTime := 0.0;
   A0302.Regolaz_Bordatrice.Formato.M1_2.Fan.Presence := FALSE;
   A0302.Regolaz_Bordatrice.Formato.M1_2.Fan.DelayOff := T#10M;
   A0302.Regolaz_Bordatrice.Formato.M1_2.Brake_Presence := FALSE;
   A0302.Regolaz_Bordatrice.Formato.M1_3.DelayMissingCondition := T#0MS;
   A0302.Regolaz_Bordatrice.Formato.M1_3.CyclicOBTime_ms := 0.0;
   A0302.Regolaz_Bordatrice.Formato.M1_3.Ax.limitMinus := 0.0;
   A0302.Regolaz_Bordatrice.Formato.M1_3.Ax.limitPlus := 0.0;
   A0302.Regolaz_Bordatrice.Formato.M1_3.Ax.Backlash := 0.0;
   A0302.Regolaz_Bordatrice.Formato.M1_3.Ax.BacklashActivation := FALSE;
   A0302.Regolaz_Bordatrice.Formato.M1_3.Ax.ToleranceWindow := 0.0;
   A0302.Regolaz_Bordatrice.Formato.M1_3.Ax.ToleranceWindowDelay := T#0MS;
   A0302.Regolaz_Bordatrice.Formato.M1_3.Ax.PreCutOff := 0.0;
   A0302.Regolaz_Bordatrice.Formato.M1_3.Ax.PreEndLowSpeed := 0.0;
   A0302.Regolaz_Bordatrice.Formato.M1_3.Ax.PreEndMedSpeed := 0.0;
   A0302.Regolaz_Bordatrice.Formato.M1_3.Ax.ChangeDirectionDelay := T#0MS;
   A0302.Regolaz_Bordatrice.Formato.M1_3.Ax.StandstillVelocity := 0.0;
   A0302.Regolaz_Bordatrice.Formato.M1_3.Ax.StandStillDelay := T#0MS;
   A0302.Regolaz_Bordatrice.Formato.M1_3.Ax.HomingDirection := FALSE;
   A0302.Regolaz_Bordatrice.Formato.M1_3.Ax.RecallTime := 0.0;
   A0302.Regolaz_Bordatrice.Formato.M1_3.Ax.VelocityFilter_T := 10.0;
   A0302.Regolaz_Bordatrice.Formato.M1_3.Ax.VelocityMeasUnit := 0;
   A0302.Regolaz_Bordatrice.Formato.M1_3.Ax.PosFbkDisabled := FALSE;
   A0302.Regolaz_Bordatrice.Formato.M1_3.Ax.FbkCtrlDisabled := FALSE;
   A0302.Regolaz_Bordatrice.Formato.M1_3.Ax_UM2."m" := 0.0;
   A0302.Regolaz_Bordatrice.Formato.M1_3.Ax_UM2.q := 0.0;
   A0302.Regolaz_Bordatrice.Formato.M1_4.DelayMissingCondition := T#0MS;
   A0302.Regolaz_Bordatrice.Formato.M1_4.CyclicOBTime_ms := 0.0;
   A0302.Regolaz_Bordatrice.Formato.M1_4.Ax.limitMinus := 0.0;
   A0302.Regolaz_Bordatrice.Formato.M1_4.Ax.limitPlus := 0.0;
   A0302.Regolaz_Bordatrice.Formato.M1_4.Ax.Backlash := 0.0;
   A0302.Regolaz_Bordatrice.Formato.M1_4.Ax.BacklashActivation := FALSE;
   A0302.Regolaz_Bordatrice.Formato.M1_4.Ax.ToleranceWindow := 0.0;
   A0302.Regolaz_Bordatrice.Formato.M1_4.Ax.ToleranceWindowDelay := T#0MS;
   A0302.Regolaz_Bordatrice.Formato.M1_4.Ax.PreCutOff := 0.0;
   A0302.Regolaz_Bordatrice.Formato.M1_4.Ax.PreEndLowSpeed := 0.0;
   A0302.Regolaz_Bordatrice.Formato.M1_4.Ax.PreEndMedSpeed := 0.0;
   A0302.Regolaz_Bordatrice.Formato.M1_4.Ax.ChangeDirectionDelay := T#0MS;
   A0302.Regolaz_Bordatrice.Formato.M1_4.Ax.StandstillVelocity := 0.0;
   A0302.Regolaz_Bordatrice.Formato.M1_4.Ax.StandStillDelay := T#0MS;
   A0302.Regolaz_Bordatrice.Formato.M1_4.Ax.HomingDirection := FALSE;
   A0302.Regolaz_Bordatrice.Formato.M1_4.Ax.RecallTime := 0.0;
   A0302.Regolaz_Bordatrice.Formato.M1_4.Ax.VelocityFilter_T := 10.0;
   A0302.Regolaz_Bordatrice.Formato.M1_4.Ax.VelocityMeasUnit := 0;
   A0302.Regolaz_Bordatrice.Formato.M1_4.Ax.PosFbkDisabled := FALSE;
   A0302.Regolaz_Bordatrice.Formato.M1_4.Ax.FbkCtrlDisabled := FALSE;
   A0302.Regolaz_Bordatrice.Formato.M1_4.Ax_UM2."m" := 0.0;
   A0302.Regolaz_Bordatrice.Formato.M1_4.Ax_UM2.q := 0.0;
   A0302.Rulliera.Ax.SLS_VEL := 3000.0;
   A0302.Rulliera.Ax.DelayMissingCondition := T#3S;
   A0302.Rulliera.Ax.Ax.SINA_Drive.ReferenceVelocity := 2200.0;
   A0302.Rulliera.Ax.Ax.SINA_Drive.InvertDirection := FALSE;
   A0302.Rulliera.Ax.Ax.MinAccTime := 0.1;
   A0302.Rulliera.Ax.Ax.MinDecTime := 0.1;
   A0302.Rulliera.Ax.Ax.LeadScrewPitchVal := 219.91;   // 359.98
   A0302.Rulliera.Ax.Ax.MotorRevolution := 6.364;
   A0302.Rulliera.Ax.Ax.LoadRevolution := 1.0;
   A0302.Rulliera.Ax.Ax.PowerOffDelay := T#1S_500MS;
   A0302.Rulliera.Ax.Ax.StandstillVelocity := 50.0;
   A0302.Rulliera.Ax.Ax.StandstillDelay := T#100MS;
   A0302.Rulliera.Ax.Fan.Presence := FALSE;
   A0302.Rulliera.Ax.Fan.DelayOff := T#0MS;
   A0302.Rulliera.Ax.Brake_Presence := FALSE;
   A0302.Centratori.Centraggio[1..3].DelayPressureRunningTimeout := T#3S;
   A0302.Centratori.Centraggio[1..3].DelayMissingCondition := T#3S;
   A0302.Centratori.Centraggio[1..3].Rest_LsQty := 1;
   A0302.Centratori.Centraggio[1..3].Work_LsQty := 0;
   A0302.Centratori.Centraggio[1..3].Rest_RetainAut := FALSE;
   A0302.Centratori.Centraggio[1..3].Work_RetainAut := FALSE;
   A0302.Centratori.Centraggio[1..3].V.RestLimSwitchExist := TRUE;
   A0302.Centratori.Centraggio[1..3].V.WorkLimSwitchExist := FALSE;
   A0302.Centratori.Centraggio[1..3].V.CheckOilInPressure := FALSE;
   A0302.Centratori.Centraggio[1..3].V.CutRestWhenIsAtRest := TRUE;
   A0302.Centratori.Centraggio[1..3].V.CutWorkWhenIsAtWork := FALSE;
   A0302.Centratori.Centraggio[1..3].V.RestTime := T#10MS;
   A0302.Centratori.Centraggio[1..3].V.WorkTime := T#300MS;
   A0302.Centratori.Centraggio[1..3].V.RestTimeOut := T#4S;
   A0302.Centratori.Centraggio[1..3].V.WorkTimeOut := T#4S;
   A0302.Centratori.Sollevamento[1..3].DelayPressureRunningTimeout := T#3S;
   A0302.Centratori.Sollevamento[1..3].DelayMissingCondition := T#3S;
   A0302.Centratori.Sollevamento[1..3].Rest_LsQty := 1;
   A0302.Centratori.Sollevamento[1..3].Work_LsQty := 1;
   A0302.Centratori.Sollevamento[1..3].Rest_RetainAut := FALSE;
   A0302.Centratori.Sollevamento[1..3].Work_RetainAut := FALSE;
   A0302.Centratori.Sollevamento[1..3].V.RestLimSwitchExist := TRUE;
   A0302.Centratori.Sollevamento[1..3].V.WorkLimSwitchExist := TRUE;
   A0302.Centratori.Sollevamento[1..3].V.CheckOilInPressure := FALSE;
   A0302.Centratori.Sollevamento[1..3].V.CutRestWhenIsAtRest := TRUE;
   A0302.Centratori.Sollevamento[1..3].V.CutWorkWhenIsAtWork := FALSE;
   A0302.Centratori.Sollevamento[1..3].V.RestTime := T#10MS;
   A0302.Centratori.Sollevamento[1..3].V.WorkTime := T#10MS;
   A0302.Centratori.Sollevamento[1..3].V.RestTimeOut := T#4S;
   A0302.Centratori.Sollevamento[1..3].V.WorkTimeOut := T#4S;
   A0302.PareggiatoreCoda.Ax.DelayMissingCondition := T#3S;
   A0302.PareggiatoreCoda.Ax.CyclicOBTime_ms := 10.0;
   A0302.PareggiatoreCoda.Ax.Ax.limitMinus := 430.0;
   A0302.PareggiatoreCoda.Ax.Ax.limitPlus := 2870.0;
   A0302.PareggiatoreCoda.Ax.Ax.Backlash := 0.0;
   A0302.PareggiatoreCoda.Ax.Ax.BacklashActivation := FALSE;
   A0302.PareggiatoreCoda.Ax.Ax.ToleranceWindow := 0.1;
   A0302.PareggiatoreCoda.Ax.Ax.ToleranceWindowDelay := T#100MS;
   A0302.PareggiatoreCoda.Ax.Ax.PreCutOff := 0.0;
   A0302.PareggiatoreCoda.Ax.Ax.PreEndLowSpeed := 0.0;
   A0302.PareggiatoreCoda.Ax.Ax.PreEndMedSpeed := 0.0;
   A0302.PareggiatoreCoda.Ax.Ax.ChangeDirectionDelay := T#0MS;
   A0302.PareggiatoreCoda.Ax.Ax.StandstillVelocity := 0.5;
   A0302.PareggiatoreCoda.Ax.Ax.StandStillDelay := T#100MS;
   A0302.PareggiatoreCoda.Ax.Ax.HomingDirection := FALSE;
   A0302.PareggiatoreCoda.Ax.Ax.RecallTime := 0.0;
   A0302.PareggiatoreCoda.Ax.Ax.VelocityFilter_T := 10.0;
   A0302.PareggiatoreCoda.Ax.Ax.VelocityMeasUnit := 2;
   A0302.PareggiatoreCoda.Ax.Ax.PosFbkDisabled := FALSE;
   A0302.PareggiatoreCoda.Ax.Ax.FbkCtrlDisabled := TRUE;
   A0302.PareggiatoreCoda.Ax.Ax_UM2."m" := 1.0;
   A0302.PareggiatoreCoda.Ax.Ax_UM2.q := -433.0;
   A0302.PareggiatoreCoda.Ax.S120.SpeedMotor.ReferenceVelocity := 2000.0;
   A0302.PareggiatoreCoda.Ax.S120.SpeedMotor.InvertDirection := FALSE;
   A0302.PareggiatoreCoda.Ax.S120.PowerOffDelay := T#5S;
   A0302.PareggiatoreCoda.Ax.S120.StandstillVelocity := 50.0;
   A0302.PareggiatoreCoda.Ax.S120.AccTime := 0.5;
   A0302.PareggiatoreCoda.Ax.S120.DecTime := 0.5;
   A0302.PareggiatoreCoda.Ax.Fan.Presence := FALSE;
   A0302.PareggiatoreCoda.Ax.Fan.DelayOff := T#10M;
   A0302.PareggiatoreCoda.Ax.Brake_Presence := FALSE;
   A0302.PareggiatoreCoda.Bloccaggio.DelayPressureRunningTimeout := T#3S;
   A0302.PareggiatoreCoda.Bloccaggio.DelayMissingCondition := T#3S;
   A0302.PareggiatoreCoda.Bloccaggio.Rest_LsQty := 1;
   A0302.PareggiatoreCoda.Bloccaggio.Work_LsQty := 1;
   A0302.PareggiatoreCoda.Bloccaggio.Rest_RetainAut := FALSE;
   A0302.PareggiatoreCoda.Bloccaggio.Work_RetainAut := FALSE;
   A0302.PareggiatoreCoda.Bloccaggio.V.RestLimSwitchExist := TRUE;
   A0302.PareggiatoreCoda.Bloccaggio.V.WorkLimSwitchExist := TRUE;
   A0302.PareggiatoreCoda.Bloccaggio.V.CheckOilInPressure := TRUE;
   A0302.PareggiatoreCoda.Bloccaggio.V.CutRestWhenIsAtRest := FALSE;
   A0302.PareggiatoreCoda.Bloccaggio.V.CutWorkWhenIsAtWork := FALSE;
   A0302.PareggiatoreCoda.Bloccaggio.V.RestTime := T#500MS;
   A0302.PareggiatoreCoda.Bloccaggio.V.WorkTime := T#500MS;
   A0302.PareggiatoreCoda.Bloccaggio.V.RestTimeOut := T#4S;
   A0302.PareggiatoreCoda.Bloccaggio.V.WorkTimeOut := T#4S;
   A0302.PareggiatoreCoda.BattutaVerticale.DelayPressureRunningTimeout := T#3S;
   A0302.PareggiatoreCoda.BattutaVerticale.DelayMissingCondition := T#3S;
   A0302.PareggiatoreCoda.BattutaVerticale.Rest_LsQty := 1;
   A0302.PareggiatoreCoda.BattutaVerticale.Work_LsQty := 1;
   A0302.PareggiatoreCoda.BattutaVerticale.Rest_RetainAut := FALSE;
   A0302.PareggiatoreCoda.BattutaVerticale.Work_RetainAut := FALSE;
   A0302.PareggiatoreCoda.BattutaVerticale.V.RestLimSwitchExist := TRUE;
   A0302.PareggiatoreCoda.BattutaVerticale.V.WorkLimSwitchExist := TRUE;
   A0302.PareggiatoreCoda.BattutaVerticale.V.CheckOilInPressure := FALSE;
   A0302.PareggiatoreCoda.BattutaVerticale.V.CutRestWhenIsAtRest := FALSE;
   A0302.PareggiatoreCoda.BattutaVerticale.V.CutWorkWhenIsAtWork := FALSE;
   A0302.PareggiatoreCoda.BattutaVerticale.V.RestTime := T#1MS;
   A0302.PareggiatoreCoda.BattutaVerticale.V.WorkTime := T#50MS;
   A0302.PareggiatoreCoda.BattutaVerticale.V.RestTimeOut := T#3S;
   A0302.PareggiatoreCoda.BattutaVerticale.V.WorkTimeOut := T#3S;
   A0302.PareggiatoreCoda.PareggiatoreLong.DelayPressureRunningTimeout := T#3S;
   A0302.PareggiatoreCoda.PareggiatoreLong.DelayMissingCondition := T#3S;
   A0302.PareggiatoreCoda.PareggiatoreLong.Rest_LsQty := 1;
   A0302.PareggiatoreCoda.PareggiatoreLong.Work_LsQty := 1;
   A0302.PareggiatoreCoda.PareggiatoreLong.Rest_RetainAut := FALSE;
   A0302.PareggiatoreCoda.PareggiatoreLong.Work_RetainAut := FALSE;
   A0302.PareggiatoreCoda.PareggiatoreLong.V.RestLimSwitchExist := TRUE;
   A0302.PareggiatoreCoda.PareggiatoreLong.V.WorkLimSwitchExist := TRUE;
   A0302.PareggiatoreCoda.PareggiatoreLong.V.CheckOilInPressure := TRUE;
   A0302.PareggiatoreCoda.PareggiatoreLong.V.CutRestWhenIsAtRest := TRUE;
   A0302.PareggiatoreCoda.PareggiatoreLong.V.CutWorkWhenIsAtWork := FALSE;
   A0302.PareggiatoreCoda.PareggiatoreLong.V.RestTime := T#500MS;
   A0302.PareggiatoreCoda.PareggiatoreLong.V.WorkTime := T#5S;
   A0302.PareggiatoreCoda.PareggiatoreLong.V.RestTimeOut := T#4S;
   A0302.PareggiatoreCoda.PareggiatoreLong.V.WorkTimeOut := T#7S;
   A0302.PareggiatoreTesta.Ax.DelayMissingCondition := T#3S;
   A0302.PareggiatoreTesta.Ax.CyclicOBTime_ms := 10.0;
   A0302.PareggiatoreTesta.Ax.Ax.limitMinus := 87.0;
   A0302.PareggiatoreTesta.Ax.Ax.limitPlus := 2502.0;
   A0302.PareggiatoreTesta.Ax.Ax.Backlash := 0.0;
   A0302.PareggiatoreTesta.Ax.Ax.BacklashActivation := FALSE;
   A0302.PareggiatoreTesta.Ax.Ax.ToleranceWindow := 0.1;
   A0302.PareggiatoreTesta.Ax.Ax.ToleranceWindowDelay := T#100MS;
   A0302.PareggiatoreTesta.Ax.Ax.PreCutOff := 0.0;
   A0302.PareggiatoreTesta.Ax.Ax.PreEndLowSpeed := 0.0;
   A0302.PareggiatoreTesta.Ax.Ax.PreEndMedSpeed := 0.0;
   A0302.PareggiatoreTesta.Ax.Ax.ChangeDirectionDelay := T#0MS;
   A0302.PareggiatoreTesta.Ax.Ax.StandstillVelocity := 0.5;
   A0302.PareggiatoreTesta.Ax.Ax.StandStillDelay := T#100MS;
   A0302.PareggiatoreTesta.Ax.Ax.HomingDirection := FALSE;
   A0302.PareggiatoreTesta.Ax.Ax.RecallTime := 0.0;
   A0302.PareggiatoreTesta.Ax.Ax.VelocityFilter_T := 10.0;
   A0302.PareggiatoreTesta.Ax.Ax.VelocityMeasUnit := 2;
   A0302.PareggiatoreTesta.Ax.Ax.PosFbkDisabled := FALSE;
   A0302.PareggiatoreTesta.Ax.Ax.FbkCtrlDisabled := TRUE;
   A0302.PareggiatoreTesta.Ax.Ax_UM2."m" := 1.0;
   A0302.PareggiatoreTesta.Ax.Ax_UM2.q := -343.0;
   A0302.PareggiatoreTesta.Ax.S120.SpeedMotor.ReferenceVelocity := 2000.0;
   A0302.PareggiatoreTesta.Ax.S120.SpeedMotor.InvertDirection := FALSE;
   A0302.PareggiatoreTesta.Ax.S120.PowerOffDelay := T#5S;
   A0302.PareggiatoreTesta.Ax.S120.StandstillVelocity := 50.0;
   A0302.PareggiatoreTesta.Ax.S120.AccTime := 0.25;
   A0302.PareggiatoreTesta.Ax.S120.DecTime := 0.25;
   A0302.PareggiatoreTesta.Ax.Fan.Presence := FALSE;
   A0302.PareggiatoreTesta.Ax.Fan.DelayOff := T#10M;
   A0302.PareggiatoreTesta.Ax.Brake_Presence := FALSE;
   A0302.PareggiatoreTesta.Bloccaggio.DelayPressureRunningTimeout := T#3S;
   A0302.PareggiatoreTesta.Bloccaggio.DelayMissingCondition := T#3S;
   A0302.PareggiatoreTesta.Bloccaggio.Rest_LsQty := 1;
   A0302.PareggiatoreTesta.Bloccaggio.Work_LsQty := 1;
   A0302.PareggiatoreTesta.Bloccaggio.Rest_RetainAut := FALSE;
   A0302.PareggiatoreTesta.Bloccaggio.Work_RetainAut := FALSE;
   A0302.PareggiatoreTesta.Bloccaggio.V.RestLimSwitchExist := TRUE;
   A0302.PareggiatoreTesta.Bloccaggio.V.WorkLimSwitchExist := TRUE;
   A0302.PareggiatoreTesta.Bloccaggio.V.CheckOilInPressure := TRUE;
   A0302.PareggiatoreTesta.Bloccaggio.V.CutRestWhenIsAtRest := FALSE;
   A0302.PareggiatoreTesta.Bloccaggio.V.CutWorkWhenIsAtWork := FALSE;
   A0302.PareggiatoreTesta.Bloccaggio.V.RestTime := T#500MS;
   A0302.PareggiatoreTesta.Bloccaggio.V.WorkTime := T#500MS;
   A0302.PareggiatoreTesta.Bloccaggio.V.RestTimeOut := T#4S;
   A0302.PareggiatoreTesta.Bloccaggio.V.WorkTimeOut := T#4S;
   A0302.PareggiatoreTesta.Sollevamento.DelayPressureRunningTimeout := T#3S;
   A0302.PareggiatoreTesta.Sollevamento.DelayMissingCondition := T#3S;
   A0302.PareggiatoreTesta.Sollevamento.Rest_LsQty := 1;
   A0302.PareggiatoreTesta.Sollevamento.Work_LsQty := 1;
   A0302.PareggiatoreTesta.Sollevamento.Rest_RetainAut := FALSE;
   A0302.PareggiatoreTesta.Sollevamento.Work_RetainAut := FALSE;
   A0302.PareggiatoreTesta.Sollevamento.V.RestLimSwitchExist := TRUE;
   A0302.PareggiatoreTesta.Sollevamento.V.WorkLimSwitchExist := TRUE;
   A0302.PareggiatoreTesta.Sollevamento.V.CheckOilInPressure := FALSE;
   A0302.PareggiatoreTesta.Sollevamento.V.CutRestWhenIsAtRest := FALSE;
   A0302.PareggiatoreTesta.Sollevamento.V.CutWorkWhenIsAtWork := FALSE;
   A0302.PareggiatoreTesta.Sollevamento.V.RestTime := T#10MS;
   A0302.PareggiatoreTesta.Sollevamento.V.WorkTime := T#10MS;
   A0302.PareggiatoreTesta.Sollevamento.V.RestTimeOut := T#5S;
   A0302.PareggiatoreTesta.Sollevamento.V.WorkTimeOut := T#5S;
   A0302.PareggiatoreTesta.Centraggio.DelayPressureRunningTimeout := T#3S;
   A0302.PareggiatoreTesta.Centraggio.DelayMissingCondition := T#3S;
   A0302.PareggiatoreTesta.Centraggio.Rest_LsQty := 1;
   A0302.PareggiatoreTesta.Centraggio.Work_LsQty := 1;
   A0302.PareggiatoreTesta.Centraggio.Rest_RetainAut := FALSE;
   A0302.PareggiatoreTesta.Centraggio.Work_RetainAut := FALSE;
   A0302.PareggiatoreTesta.Centraggio.V.RestLimSwitchExist := TRUE;
   A0302.PareggiatoreTesta.Centraggio.V.WorkLimSwitchExist := FALSE;
   A0302.PareggiatoreTesta.Centraggio.V.CheckOilInPressure := FALSE;
   A0302.PareggiatoreTesta.Centraggio.V.CutRestWhenIsAtRest := FALSE;
   A0302.PareggiatoreTesta.Centraggio.V.CutWorkWhenIsAtWork := FALSE;
   A0302.PareggiatoreTesta.Centraggio.V.RestTime := T#10MS;
   A0302.PareggiatoreTesta.Centraggio.V.WorkTime := T#10MS;
   A0302.PareggiatoreTesta.Centraggio.V.RestTimeOut := T#5S;
   A0302.PareggiatoreTesta.Centraggio.V.WorkTimeOut := T#5S;
   A0302.Manipolatore.Testa.Ax.SLS_Vel := 3000.0;
   A0302.Manipolatore.Testa.Ax.DelayMissingCondition := T#1S;
   A0302.Manipolatore.Testa.Ax.Ax.Encoder_Inc_AutoReloadPosition := FALSE;
   A0302.Manipolatore.Testa.Ax.Ax.Encoder_is_Absolute := TRUE;
   A0302.Manipolatore.Testa.Ax.Ax.LeadScrewPitchVal := 10.4992026;
   A0302.Manipolatore.Testa.Ax.Ax.MotorRevolution := 66.84;
   A0302.Manipolatore.Testa.Ax.Ax.LoadRevolution := 1.0;
   A0302.Manipolatore.Testa.Ax.Ax.PowerOffDelay := T#500MS;
   A0302.Manipolatore.Testa.Ax.Ax.MaxRPM_S120_P2000 := 8000.0;
   A0302.Manipolatore.Testa.Ax.Ax.MaxVel_S120_P2571 := 31500.0;
   A0302.Manipolatore.Testa.Ax.Ax.MaxAcc_S120_P2572 := 2000.0;
   A0302.Manipolatore.Testa.Ax.Ax.MaxDec_S120_P2573 := 2000.0;
   A0302.Manipolatore.Testa.Ax.Ax.Modulo_S120_P2566 := 0.0;
   A0302.Manipolatore.Testa.Ax.Ax.SwLimMinus_S120_P2580 := -650.0;
   A0302.Manipolatore.Testa.Ax.Ax.SwLimPlus_S120_P2581 := 553.0;
   A0302.Manipolatore.Testa.Ax.Fan.Presence := FALSE;
   A0302.Manipolatore.Testa.Ax.Fan.DelayOff := T#0MS;
   A0302.Manipolatore.Testa.Ax.Brake_Presence := FALSE;
   A0302.Manipolatore.Testa.Sollevatore.DelayPressureRunningTimeout := T#3S;
   A0302.Manipolatore.Testa.Sollevatore.DelayMissingCondition := T#3S;
   A0302.Manipolatore.Testa.Sollevatore.Rest_LsQty := 1;
   A0302.Manipolatore.Testa.Sollevatore.Work_LsQty := 0;
   A0302.Manipolatore.Testa.Sollevatore.Rest_RetainAut := FALSE;
   A0302.Manipolatore.Testa.Sollevatore.Work_RetainAut := FALSE;
   A0302.Manipolatore.Testa.Sollevatore.V.RestLimSwitchExist := TRUE;
   A0302.Manipolatore.Testa.Sollevatore.V.WorkLimSwitchExist := FALSE;
   A0302.Manipolatore.Testa.Sollevatore.V.CheckOilInPressure := FALSE;
   A0302.Manipolatore.Testa.Sollevatore.V.CutRestWhenIsAtRest := FALSE;
   A0302.Manipolatore.Testa.Sollevatore.V.CutWorkWhenIsAtWork := FALSE;
   A0302.Manipolatore.Testa.Sollevatore.V.RestTime := T#1MS;
   A0302.Manipolatore.Testa.Sollevatore.V.WorkTime := T#200MS;
   A0302.Manipolatore.Testa.Sollevatore.V.RestTimeOut := T#5S;
   A0302.Manipolatore.Testa.Sollevatore.V.WorkTimeOut := T#5S;
   A0302.Manipolatore.Testa.Magnete.DelayPressureRunningTimeout := T#3S;
   A0302.Manipolatore.Testa.Magnete.DelayMissingCondition := T#3S;
   A0302.Manipolatore.Testa.Magnete.Rest_LsQty := 1;
   A0302.Manipolatore.Testa.Magnete.Work_LsQty := 0;
   A0302.Manipolatore.Testa.Magnete.Rest_RetainAut := FALSE;
   A0302.Manipolatore.Testa.Magnete.Work_RetainAut := FALSE;
   A0302.Manipolatore.Testa.Magnete.V.RestLimSwitchExist := TRUE;
   A0302.Manipolatore.Testa.Magnete.V.WorkLimSwitchExist := FALSE;
   A0302.Manipolatore.Testa.Magnete.V.CheckOilInPressure := FALSE;
   A0302.Manipolatore.Testa.Magnete.V.CutRestWhenIsAtRest := TRUE;
   A0302.Manipolatore.Testa.Magnete.V.CutWorkWhenIsAtWork := FALSE;
   A0302.Manipolatore.Testa.Magnete.V.RestTime := T#1MS;
   A0302.Manipolatore.Testa.Magnete.V.WorkTime := T#300MS;
   A0302.Manipolatore.Testa.Magnete.V.RestTimeOut := T#5S;
   A0302.Manipolatore.Testa.Magnete.V.WorkTimeOut := T#5S;
   A0302.Manipolatore.Coda.Ax.SLS_Vel := 3000.0;
   A0302.Manipolatore.Coda.Ax.DelayMissingCondition := T#1S;
   A0302.Manipolatore.Coda.Ax.Ax.Encoder_Inc_AutoReloadPosition := FALSE;
   A0302.Manipolatore.Coda.Ax.Ax.Encoder_is_Absolute := TRUE;
   A0302.Manipolatore.Coda.Ax.Ax.LeadScrewPitchVal := 10.4992026;
   A0302.Manipolatore.Coda.Ax.Ax.MotorRevolution := 66.84;
   A0302.Manipolatore.Coda.Ax.Ax.LoadRevolution := 0.0;
   A0302.Manipolatore.Coda.Ax.Ax.PowerOffDelay := T#0MS;
   A0302.Manipolatore.Coda.Ax.Ax.MaxRPM_S120_P2000 := 8000.0;
   A0302.Manipolatore.Coda.Ax.Ax.MaxVel_S120_P2571 := 31500.0;
   A0302.Manipolatore.Coda.Ax.Ax.MaxAcc_S120_P2572 := 2000.0;
   A0302.Manipolatore.Coda.Ax.Ax.MaxDec_S120_P2573 := 2000.0;
   A0302.Manipolatore.Coda.Ax.Ax.Modulo_S120_P2566 := 0.0;
   A0302.Manipolatore.Coda.Ax.Ax.SwLimMinus_S120_P2580 := -650.0;
   A0302.Manipolatore.Coda.Ax.Ax.SwLimPlus_S120_P2581 := 552.0;
   A0302.Manipolatore.Coda.Ax.Fan.Presence := FALSE;
   A0302.Manipolatore.Coda.Ax.Fan.DelayOff := T#0MS;
   A0302.Manipolatore.Coda.Ax.Brake_Presence := FALSE;
   A0302.Manipolatore.Coda.Sollevatore.DelayPressureRunningTimeout := T#3S;
   A0302.Manipolatore.Coda.Sollevatore.DelayMissingCondition := T#3S;
   A0302.Manipolatore.Coda.Sollevatore.Rest_LsQty := 1;
   A0302.Manipolatore.Coda.Sollevatore.Work_LsQty := 0;
   A0302.Manipolatore.Coda.Sollevatore.Rest_RetainAut := FALSE;
   A0302.Manipolatore.Coda.Sollevatore.Work_RetainAut := FALSE;
   A0302.Manipolatore.Coda.Sollevatore.V.RestLimSwitchExist := TRUE;
   A0302.Manipolatore.Coda.Sollevatore.V.WorkLimSwitchExist := FALSE;
   A0302.Manipolatore.Coda.Sollevatore.V.CheckOilInPressure := FALSE;
   A0302.Manipolatore.Coda.Sollevatore.V.CutRestWhenIsAtRest := FALSE;
   A0302.Manipolatore.Coda.Sollevatore.V.CutWorkWhenIsAtWork := FALSE;
   A0302.Manipolatore.Coda.Sollevatore.V.RestTime := T#1MS;
   A0302.Manipolatore.Coda.Sollevatore.V.WorkTime := T#200MS;
   A0302.Manipolatore.Coda.Sollevatore.V.RestTimeOut := T#5S;
   A0302.Manipolatore.Coda.Sollevatore.V.WorkTimeOut := T#5S;
   A0302.Manipolatore.Coda.Magnete.DelayPressureRunningTimeout := T#3S;
   A0302.Manipolatore.Coda.Magnete.DelayMissingCondition := T#3S;
   A0302.Manipolatore.Coda.Magnete.Rest_LsQty := 1;
   A0302.Manipolatore.Coda.Magnete.Work_LsQty := 0;
   A0302.Manipolatore.Coda.Magnete.Rest_RetainAut := FALSE;
   A0302.Manipolatore.Coda.Magnete.Work_RetainAut := FALSE;
   A0302.Manipolatore.Coda.Magnete.V.RestLimSwitchExist := TRUE;
   A0302.Manipolatore.Coda.Magnete.V.WorkLimSwitchExist := FALSE;
   A0302.Manipolatore.Coda.Magnete.V.CheckOilInPressure := FALSE;
   A0302.Manipolatore.Coda.Magnete.V.CutRestWhenIsAtRest := TRUE;
   A0302.Manipolatore.Coda.Magnete.V.CutWorkWhenIsAtWork := FALSE;
   A0302.Manipolatore.Coda.Magnete.V.RestTime := T#1MS;
   A0302.Manipolatore.Coda.Magnete.V.WorkTime := T#300MS;
   A0302.Manipolatore.Coda.Magnete.V.RestTimeOut := T#5S;
   A0302.Manipolatore.Coda.Magnete.V.WorkTimeOut := T#5S;
END_DATA_BLOCK

DATA_BLOCK "Area03_Messages"   // DB108
// stored: MemoryReserve 100
   VAR
      "A" : Struct
         Msg : Array[1..736] of Bool;
         Hmi : Array[1..46] of Word;
         Ack : Array[1..46] of Word;
      END_STRUCT;
      W : Struct
         Msg : Array[1..832] of Bool;
         Hmi : Array[1..52] of Word;
         Ack : Array[1..52] of Word;
      END_STRUCT;
   END_VAR
BEGIN
   // "A".Msg[2] : h
   // "A".Msg[3] : hsfdd
END_DATA_BLOCK

DATA_BLOCK "A03_HMI"   // DB78
// stored: MemoryReserve 0
   VAR
      Area03 : Struct
         Status : "StatusArea";
         SuperUser : "SuperUser";
      END_STRUCT;
      MB3 : Struct
         ManCode_REQ : Int;
         ManCode_CMD : Int;
         Button : Struct
            A0301 : Struct
               Trasporto : "Ax_PB";
               Ribaltatore : Struct
                  Solleva_Rib : "ValveMachine_PB";
                  Rotazione : "Ax_PB";
               END_STRUCT;
               P1 : Struct
                  Fermi : "ValveMachine_PB";
                  Pareggiatore : "ValveMachine_PB";
               END_STRUCT;
               P2 : Struct
                  Fermi : "ValveMachine_PB";
                  Sollevatori : "ValveMachine_PB";
               END_STRUCT;
               P3 : Struct
                  Fermi : "ValveMachine_PB";
               END_STRUCT;
               P4 : Struct
                  Fermi : "ValveMachine_PB";
               END_STRUCT;
               SpintoreLat : Struct
                  OP : "OP_PB";
                  Vrt : "ValveMachine_PB";
                  Orz : "ValveMachine_PB";
                  Sollevatori : "ValveMachine_PB";
               END_STRUCT;
            END_STRUCT;
            A0302 : Struct
               HU_Cytropack : Struct
                  Start : Bool;
                  Stop : Bool;
               END_STRUCT;
               SpintoreLong : Struct
                  OP : "OP_PB";
                  Ax : "Ax_PB";
                  Vrt : "ValveMachine_PB";
                  Orz : "ValveMachine_PB";
               END_STRUCT;
               Bordatrice : Struct
                  OP_Ax : "Ax_PB";
                  Ax : "Ax_PB";
                  Regolazione : Struct
                     Single_PB : Array[1..10] of "Ax_PB";
                     Passaggio_Combo : Array[1..4] of "Ax_PB";
                     Ax : "Ax_PB";
                  END_STRUCT;
               END_STRUCT;
               Rulliera : Struct   // Con selezione delle 2
                  OP : "OP_PB";   // REST NON C'E
                  Ax : "Ax_PB";   // POS NON C'E
               END_STRUCT;
               Centratori : Struct   // Con selezione dei 4
                  OP { S7_SetPoint := 'True'} : "OP_PB";
                  Centraggio : "ValveMachine_PB";
                  Sollevamento : "ValveMachine_PB";
               END_STRUCT;
               PareggiatoreCoda : Struct
                  OP_Ax : "Ax_PB";
                  OP_BattutaVrt : "OP_PB";
                  OP_PareggLong : "OP_PB";
                  Ax : "Ax_PB";
                  Bloccaggio : "ValveMachine_PB";
                  BattutaVerticale : "ValveMachine_PB";
                  PareggiatoreLongitudinale : "ValveMachine_PB";
               END_STRUCT;
               PareggiatoreTesta : Struct
                  OP_Ax : "Ax_PB";
                  OP_Sollevamento : "OP_PB";
                  OP_Centraggio : "OP_PB";
                  Ax : "Ax_PB";
                  Bloccaggio : "ValveMachine_PB";
                  Centratore : "ValveMachine_PB";
                  Sollevamento : "ValveMachine_PB";
               END_STRUCT;
               Manipolatore : Struct   // Con selezione testa coda
                  OP_Ax : Struct
                     MoveToPos : Bool;
                  END_STRUCT;
                  OP_Sollevamento : "OP_PB";
                  OP_Magneti : "OP_PB";
                  Ax : "Ax_PB";
                  Sollevatore : "ValveMachine_PB";
                  Magnete : "ValveMachine_PB";
               END_STRUCT;
            END_STRUCT;
            A0303 : Struct
               Spalla : Struct
                  Testa : Struct
                     OP_Pos : Bool;
                     Ax : "Ax_PB";
                  END_STRUCT;
                  Coda : Struct
                     OP_Pos : Bool;
                     Ax : "Ax_PB";
                  END_STRUCT;
               END_STRUCT;
               SpintoreStrato : Struct   // Con selezione testa coda
                  OP_Work : Bool;
                  OP_Rest : Bool;
                  Vrt : "ValveMachine_PB";
                  Orz : "ValveMachine_PB";
               END_STRUCT;
               TraslazioneStrato : Struct   // Con selezione testa coda
                  OP_Vai_A_Prelievo : Bool;
                  OP_Prelievo : Bool;
                  OP_Vai_A_Deposito : Bool;
                  OP_Deposito : Bool;
                  Ax : "Ax_PB";
                  Manip_Sostegno : "ValveMachine_PB";
                  Manip_Pareggiatore : "ValveMachine_PB";
                  SostegnoVrt { S7_SetPoint := 'True'} : "ValveMachine_PB";
               END_STRUCT;
               SollevamentoStrato : Struct   // Con selezione testa coda
                  OP_Prelievo : Bool;
                  OP_Deposito : Bool;
                  Ax : "Ax_PB";   // Con selezione testa coda
               END_STRUCT;
               SostegnoAntirib : Struct   // Con selezione testa coda
                  Testa : Struct
                     OP_Ax : Struct
                        MoveToPos : Bool;
                     END_STRUCT;
                     OP_Paletti : Struct
                        Rest : Bool;
                        Work : Bool;
                     END_STRUCT;
                     Ax : "Ax_PB";
                     Paletti : Struct
                        Pos0 { S7_SetPoint := 'True'} : Bool;
                        Pos1 : Bool;
                        Pos2 : Bool;
                     END_STRUCT;
                  END_STRUCT;
                  Coda : Struct
                     OP_Ax : Struct
                        MoveToPos : Bool;
                     END_STRUCT;
                     OP_Paletti : Struct
                        Rest : Bool;
                        Work : Bool;
                     END_STRUCT;
                     Ax : "Ax_PB";
                     Paletti : Struct
                        Pos0 { S7_SetPoint := 'True'} : Bool;
                        Pos1 : Bool;
                        Pos2 : Bool;
                     END_STRUCT;
                  END_STRUCT;
               END_STRUCT;
            END_STRUCT;
            A0304 : Struct
               Navetta : Struct   // Con selezione e op
                  OP_Vai_A_Prelievo : Bool;
                  OP_Prelievo : Bool;
                  OP_Vai_A_Deposito : Bool;
                  Ax : "Ax_PB";
                  Paletti : Struct   // Con selezione
                     Esterni : "ValveMachine_PB";
                     Interni : "ValveMachine_PB";
                  END_STRUCT;
               END_STRUCT;
            END_STRUCT;
            PB_Empty : Struct
               Valve { S7_SetPoint := 'True'} : "ValveMachine_PB";
               Ax { S7_SetPoint := 'True'} : "Ax_PB";
            END_STRUCT;
         END_STRUCT;
      END_STRUCT;
   END_VAR
BEGIN
END_DATA_BLOCK

DATA_BLOCK "A0301_PERS"   // DB41
// stored: MemoryReserve 100
   VAR RETAIN
      Par : Struct
         Maint_FreeMove : Bool := FALSE;   // Manutenzione: movimento libero
         CaseA_PLen_Lim : Real := 700.0;   // [mm] Caso A : Lunghezza SG limite (da 900 a..)
         CaseA_StopperSensor : USInt := 1;   // Caso A : Sensori da usare su stopper
         CaseB_PLen_Lim : Real := 1990.0;   // [mm] Caso B : Lunghezza SG limite (da 900 a..)
         CaseB_StopperSensor : USInt := 3;   // Caso B : Sensori da usare su stopper
         CaseC_PLen_Lim : Real := 2000.0;   // [mm] Caso C : Lunghezza SG limite (da 900 a..)
         CaseC_StopperSensor : USInt := 3;   // Caso C : Sensori da usare su stopper
         CaseD_PLen_Lim : Real := 2100.0;   // [mm] Caso D : Lunghezza SG limite A (da 900 a..)
         CaseD_StopperSensor : USInt := 3;   // Caso D : Sensori da usare su stopper
         DlySensorsON { S7_SetPoint := 'True'} : Time := T#1S;   // [ms] Ritrado ON sensori prima e dopo fermi
         DlySensorsOFF { S7_SetPoint := 'True'} : Time := T#1S;   // [ms] Ritrado OFF sensori prima e dopo fermi
         TolReachNextStopper : Real := 70.0;   // [mm] Tolleranza movimento SG su stopper (Almeno un sensore in uso ON)
         TolReachAllSensorsON : Real := 50.0;   // [mm] Tolleranza posizione raggiunta (Sensori in uso ON)
      END_STRUCT;
      Par_Mng : Struct
         DlySensorsON { S7_SetPoint := 'True'} : Time := T#1S;   // [ms] Ritrado ON sensori prima e dopo fermi
         DlySensorsOFF { S7_SetPoint := 'True'} : Time := T#1S;   // [ms] Ritrado OFF sensori prima e dopo fermi
         TRK : Struct
            BTrk_MoveP4Exit { S7_SetPoint := 'True'} : Time := T#500MS;
            BTrk_MoveToP5 { S7_SetPoint := 'True'} : Time := T#500MS;
         END_STRUCT;
      END_STRUCT;
      Data_Mng { ExternalWritable := 'False'} : Struct
         LastCounter_PartMove_P2toP4 : LReal := 999999.999999998;
         LastCounter_PartMove_P1toP2 : LReal := 999999.999999998;
         LastCounter_PartMove_P1toP3 : LReal := 2.50784669856199;
      END_STRUCT;
   END_VAR
   VAR
      FC_Sensor : Struct
         "Case" : Int := 1;
      END_STRUCT;
   END_VAR
   VAR RETAIN
      SensTime : Struct
         P1 : Struct
            Sens_Ing : Struct
               DelayOn : Time := T#500MS;
            END_STRUCT;
            Sens_Out : Struct
               DelayOff : Time := T#300MS;
            END_STRUCT;
         END_STRUCT;
         P2 : Struct
            Sens_Ing : Struct
               DelayOn : Time := T#100MS;
            END_STRUCT;
            Sens_Out : Struct
               DelayOff : Time := T#500MS;
            END_STRUCT;
         END_STRUCT;
         P3 : Struct
            Sens_Ing : Struct
               DelayOn : Time := T#100MS;
            END_STRUCT;
            Sens_Out : Struct
               DelayOff : Time := T#100MS;
            END_STRUCT;
         END_STRUCT;
         P4 : Struct
            Sens_Ing : Struct
               DelayOn : Time := T#100MS;
            END_STRUCT;
            Sens_Out : Struct
               DelayOff : Time := T#100MS;
            END_STRUCT;
         END_STRUCT;
      END_STRUCT;
   END_VAR
BEGIN
END_DATA_BLOCK

DATA_BLOCK "A0301_Trasporto_PERS"   // DB37
// stored: MemoryReserve 100
   VAR RETAIN
      Par : Struct
         Ax { S7_SetPoint := 'True'} : "SpeedMachine_Par";
         Ax_Aut { S7_SetPoint := 'True'} : "A0301_Mach_Speed_Par";
      END_STRUCT;
   END_VAR
BEGIN
   Par.Ax.Man.VelBwd := 10000.0;
   Par.Ax.Man.VelFwdHigh := 10000.0;
   Par.Ax.Man.VelFwdLow := 10000.0;
   Par.Ax.Man.Acc := 1000.0;
   Par.Ax.Man.Dec := 1000.0;
   Par.Ax.Man.DelayChangeVel := T#100MS;
   Par.Ax_Aut.SemiAut_Vel := 15000.0;
   Par.Ax_Aut.Aut_Vel := 20000.0;
   Par.Ax_Aut.Aut_Acc := 1500.0;
   Par.Ax_Aut.Aut_Dec := 1500.0;
END_DATA_BLOCK

DATA_BLOCK "A0301_Ribaltatore_PERS"   // DB58
// stored: MemoryReserve 100
   VAR RETAIN
      Par_Manu : "Positioning_EPOS_Machine_Par";
      Par_Aut : "A0301_Mach_Ribaltatore_Par";
   END_VAR
   VAR
      Par_Aut_Vel : Struct
         Pos1_Frw : LReal := 5000.0;
         Pos2_Frw : LReal := 5000.0;
         Pos0_Brw : LReal := 60000.0;
      END_STRUCT;
   END_VAR
   VAR RETAIN
      Pers_Data : Struct
         EncoderAbsolute_Preset_OK : Bool := TRUE;
         Persistent_ActualPosition : LReal := 2.0;
      END_STRUCT;
   END_VAR
BEGIN
   Par_Manu.PosTolerance := 0.5;
   Par_Manu.DelayInPosition := T#100MS;
   Par_Manu.Man_Vel := 15000.0;
   Par_Manu.Man_Acc := 1000.0;
   Par_Manu.Man_Dec := 1000.0;
   Par_Aut.SemiAut_Vel := 8000.0;
   Par_Aut.Aut_Vel := 8000.0;
   Par_Aut.Aut_Acc := 1000.0;
   Par_Aut.Aut_Dec := 1000.0;
   Par_Aut.Pos_0 := 2.0;
   Par_Aut.Pos_1 := 40.0;
   Par_Aut.Pos_2 := 70.0;
   Par_Aut.Pos_3 := 120.0;
END_DATA_BLOCK

DATA_BLOCK "A0301_Spintore_Lat_PERS"   // DB35
// stored: MemoryReserve 100
   VAR RETAIN
      Spin_Lat_1 : Struct
         Par { S7_SetPoint := 'True'} : "Analogic_SensorManagement_Par";
         Data : Struct
            Sens { S7_SetPoint := 'True'} : "Analogic_SensorManagement_Data";
            HMI { ExternalAccessible := 'False'; ExternalVisible := 'False'; ExternalWritable := 'False'} : "HMI_Preset";
         END_STRUCT;
         Par_Mach { S7_SetPoint := 'True'} : "A0301_Mach_Sens_Par";
      END_STRUCT;
      Spin_Lat_2 : Struct
         Par : "Analogic_SensorManagement_Par";
         Data : Struct
            Sens { S7_SetPoint := 'True'} : "Analogic_SensorManagement_Data";
            HMI : "HMI_Preset";
         END_STRUCT;
         Par_Mach : "A0301_Mach_Sens_Par";
      END_STRUCT;
   END_VAR
BEGIN
   Spin_Lat_1.Par.Enable := TRUE;   // 1= Enable / 0 Disable
   Spin_Lat_1.Par.RangeLow := 260.0;   // Corsa minima pistone
   Spin_Lat_1.Par.RangeHigh := 60.0;   // Corsa massima pistone
   Spin_Lat_1.Data.Sens.OffsetValue := 5.88212585449219;   // Valore aggiunto o sottratto a Out.ScaleValue
   Spin_Lat_1.Data.Sens.OffsetValid := TRUE;   // Stato di ritorno del valore offset
   Spin_Lat_1.Data.HMI.Button := FALSE;
   Spin_Lat_1.Data.HMI.Value := 260.0;
   Spin_Lat_1.Data.HMI.Feedback := 260.029876708984;
   Spin_Lat_1.Par_Mach.Tol_Work := 180.0;
   Spin_Lat_1.Par_Mach.WorkTime_SensDisable := T#100MS;
   Spin_Lat_2.Par.Enable := TRUE;   // 1= Enable / 0 Disable
   Spin_Lat_2.Par.RangeLow := 260.0;   // Corsa minima pistone
   Spin_Lat_2.Par.RangeHigh := 60.0;   // Corsa massima pistone
   Spin_Lat_2.Data.Sens.OffsetValue := 6.43084716796875;   // Valore aggiunto o sottratto a Out.ScaleValue
   Spin_Lat_2.Data.Sens.OffsetValid := TRUE;   // Stato di ritorno del valore offset
   Spin_Lat_2.Data.HMI.Button := FALSE;
   Spin_Lat_2.Data.HMI.Value := 260.0;
   Spin_Lat_2.Data.HMI.Feedback := 260.0;
   Spin_Lat_2.Par_Mach.Tol_Work := 180.0;
   Spin_Lat_2.Par_Mach.WorkTime_SensDisable := T#100MS;
END_DATA_BLOCK

DATA_BLOCK "A0302_PERS"   // DB107
// stored: MemoryReserve 100
   VAR RETAIN
      Par : Struct
         CarroPareggCoda : Struct
            Delay_StartMove : Time;
            Preset { S7_SetPoint := 'True'} : LReal := 435.433;
         END_STRUCT;
         CarroPareggTesta : Struct
            Delay_StartMove : Time;
            Preset { S7_SetPoint := 'True'} : LReal := 348.633;
         END_STRUCT;
         Cremaliera : Struct
            Modulo { S7_SetPoint := 'True'} : LReal := 2.5;
            Passo { S7_SetPoint := 'True'} : LReal := 7.854;
         END_STRUCT;
      END_STRUCT;
   END_VAR
BEGIN
END_DATA_BLOCK

DATA_BLOCK "A0302_HU_Cytropack_PERS"   // DB195
// stored: MemoryReserve 100
   VAR RETAIN
      Par : Struct
         Bloccaggio : Struct
            TargetPressure : Real := 100.0;
            TargetMaxSpeed : Real := 3000.0;
            Delta : Struct
               Min : Real := 0.5;
               Max : Real := 0.5;
            END_STRUCT;
         END_STRUCT;
         Pareggiamento : Struct
            TargetPressure : Real := 100.0;
            TargetMaxSpeed : Real := 3000.0;
            Delta : Struct
               Min : Real := 0.5;
               Max : Real := 0.5;
            END_STRUCT;
         END_STRUCT;
      END_STRUCT;
   END_VAR
BEGIN
END_DATA_BLOCK

DATA_BLOCK "A0302_Spintore_PERS"   // DB76
// stored: MemoryReserve 100
   VAR RETAIN
      Par : Struct
         Sens : "Analogic_SensorManagement_Par";
      END_STRUCT;
      Data : Struct
         Sens : "Analogic_SensorManagement_Data";
         HMI { ExternalAccessible := 'False'; ExternalVisible := 'False'; ExternalWritable := 'False'} : "HMI_Preset";
         Ax_Pos : "A0301_Mach_Ax_Pos_Data";
      END_STRUCT;
      Par_Mach { S7_SetPoint := 'True'} : "A0301_Mach_Sens_Par";
      Par_Ax_Manu : "Positioning_EPOS_Machine_Par";
      Pers_Data : Struct
         EncoderAbsolute_Preset_OK : Bool := TRUE;
         Persistent_ActualPosition : LReal := 670.75;
      END_STRUCT;
      Par_Ax_Auto : "A0301_Mach_Speed_Par";
   END_VAR
BEGIN
   Par.Sens.Enable := TRUE;
   Par.Sens.RangeLow := 0.0;
   Par.Sens.RangeHigh := 150.0;
   Data.Sens.OffsetValue := 18.9832916259766;
   Data.Sens.OffsetValid := TRUE;
   Data.HMI.Button := FALSE;
   Data.HMI.Value := 150.0;
   Data.HMI.Feedback := 150.037933349609;
   Data.Ax_Pos.OffsetPosAttesa := 500.0;
   Data.Ax_Pos.PosAttesa := 670.75;
   Data.Ax_Pos.PosFineSpinta := 1170.75;
   Par_Mach.Tol_Work := 100.0;
   Par_Mach.WorkTime_SensDisable := T#100MS;
   Par_Ax_Manu.PosTolerance := 0.5;
   Par_Ax_Manu.DelayInPosition := T#10MS;
   Par_Ax_Manu.Man_Vel := 20000.0;
   Par_Ax_Manu.Man_Acc := 3000.0;
   Par_Ax_Manu.Man_Dec := 1000.0;
   Par_Ax_Auto.SemiAut_Vel := 25000.0;
   Par_Ax_Auto.Aut_Vel := 20000.0;
   Par_Ax_Auto.Aut_Acc := 3000.0;
   Par_Ax_Auto.Aut_Dec := 1000.0;
END_DATA_BLOCK

DATA_BLOCK "A0302_PareggiatoreCoda_PERS"   // DB120
// stored: MemoryReserve 100
   VAR RETAIN
      Par : Struct
         Ax { S7_SetPoint := 'True'} : "Positioning_DOL_Machine_Par";
         Ax_Pers { ExternalAccessible := 'False'; ExternalVisible := 'False'; ExternalWritable := 'False'} : "Positioning_DOL_Machine_Pers_Data";
         Enc : "PosFbk_RTN";
         Ax_Aut { S7_SetPoint := 'True'} : "A0301_Mach_Speed_Par";
         Bloccaggio_Sens : Struct
            "2191B1" : "Analogic_SensorManagement_Par";
            SogliaWork { S7_SetPoint := 'True'} : Real := 0.0;
         END_STRUCT;
         CarroPareggCoda : Struct
            Delay_StartMove : Time := T#100MS;
            Preset { S7_SetPoint := 'True'} : LReal := 477.68;
         END_STRUCT;
         Cremaliera : Struct
            Modulo { S7_SetPoint := 'True'} : LReal := 2.5;
            Passo { S7_SetPoint := 'True'} : LReal := 7.854;
         END_STRUCT;
      END_STRUCT;
      Par_Sens : Struct
         AI { S7_SetPoint := 'True'} : "Analogic_SensorManagement_Par";
      END_STRUCT;
      Data_Sens { S7_SetPoint := 'True'} : "Analogic_SensorManagement_Data";
      Par_MachSens { S7_SetPoint := 'True'} : "A0301_Mach_Sens_Par";
      IEC_SP : Struct
         FTC_Input : Struct
            TON_PT : Time := T#10MS;
            TOF_PT : Time := T#100MS;
         END_STRUCT;
         FTC_Output : Struct
            TON_PT : Time := T#10MS;
            TOF_PT : Time := T#10MS;
         END_STRUCT;
         FTC_PresentMat : Struct
            TON_PT : Time := T#500MS;
            TOF_PT : Time := T#500MS;
         END_STRUCT;
         Check_2119B1 { ExternalAccessible := 'False'; ExternalVisible := 'False'; ExternalWritable := 'False'} : Struct
            TON_PT : Time := T#500MS;
         END_STRUCT;
      END_STRUCT;
   END_VAR
BEGIN
   Par.Ax.PosTolerance := 1.0;
   Par.Ax.Minus_Limit := 457.6;
   Par.Ax.Plus_Limit := 2845.0;
   Par.Ax.PreCutOff := 0.2;
   Par.Ax.PreEndLowSpeed := 2.0;
   Par.Ax.PreEndMedSpeed := 5.0;
   Par.Ax.LowSpeed := 2.0;
   Par.Ax.MedSpeed := 5.0;
   Par.Ax.HighSpeed := 50.0;
   Par.Ax.Man_Speed := 50.0;
   Par.Ax_Pers.AxisHomed := TRUE;
   Par.Enc.Preset.Pulses := 1_666_530_232;
   Par.Enc.Preset.Units := 477.68;
   Par.Enc.Config.Resolution := 125.663706143592;
   Par.Ax_Aut.SemiAut_Vel := 50.0;
   Par.Ax_Aut.Aut_Vel := 50.0;
   Par.Ax_Aut.Aut_Acc := 1.0;
   Par.Ax_Aut.Aut_Dec := 1.0;
   Par.Bloccaggio_Sens."2191B1".Enable := TRUE;
   Par.Bloccaggio_Sens."2191B1".RangeLow := 0.0;
   Par.Bloccaggio_Sens."2191B1".RangeHigh := 0.0;
   Par_Sens.AI.Enable := TRUE;
   Par_Sens.AI.RangeLow := 43.0;
   Par_Sens.AI.RangeHigh := 133.7;
   Data_Sens.OffsetValue := -4.04816818237305;
   Data_Sens.OffsetValid := TRUE;
   Par_MachSens.Tol_Work := 89.3;
   Par_MachSens.WorkTime_SensDisable := T#10MS;
END_DATA_BLOCK

DATA_BLOCK "A0302_PareggiatoreTesta_PERS"   // DB123
// stored: MemoryReserve 100
   VAR RETAIN
      Par : Struct
         Ax : "Positioning_DOL_Machine_Par";
         Ax_Pers { ExternalAccessible := 'False'; ExternalVisible := 'False'; ExternalWritable := 'False'} : "Positioning_DOL_Machine_Pers_Data";
         Enc : "PosFbk_RTN";
         Ax_Aut : "A0301_Mach_Speed_Par";
         Bloccaggio_Sens : Struct
            "2111B1" : "Analogic_SensorManagement_Par";
            SogliaWork : Real := 0.0;
         END_STRUCT;
         CarroPareggTesta { ExternalAccessible := 'False'; ExternalVisible := 'False'; ExternalWritable := 'False'} : Struct
            Delay_StartMove : Time := T#100MS;
            Preset : LReal := 348.5;
         END_STRUCT;
         Cremaliera { ExternalAccessible := 'False'; ExternalVisible := 'False'; ExternalWritable := 'False'} : Struct
            Modulo : LReal := 2.5;
            Passo : LReal := 7.854;
         END_STRUCT;
      END_STRUCT;
      IEC_SP : Struct
         FTC_Rall : Struct
            TON_PT : Time := T#1MS;
            TOF_PT : Time := T#200MS;
         END_STRUCT;
         FTC_ProxLs : Struct
            TON_PT : Time := T#1MS;
            TOF_PT : Time := T#200MS;
         END_STRUCT;
         FTC_PresentMat : Struct
            TON_PT : Time := T#500MS;
            TOF_PT : Time := T#500MS;
         END_STRUCT;
         Check_2111B1 : Struct
            TON_PT : Time := T#500MS;
         END_STRUCT;
      END_STRUCT;
   END_VAR
BEGIN
   Par.Ax.PosTolerance := 0.5;
   Par.Ax.Minus_Limit := 338.5;
   Par.Ax.Plus_Limit := 2770.0;
   Par.Ax.PreCutOff := 0.2;
   Par.Ax.PreEndLowSpeed := 2.0;
   Par.Ax.PreEndMedSpeed := 5.0;
   Par.Ax.LowSpeed := 5.0;
   Par.Ax.MedSpeed := 10.0;
   Par.Ax.HighSpeed := 70.0;
   Par.Ax.Man_Speed := 20.0;
   Par.Ax_Pers.AxisHomed := TRUE;
   Par.Enc.Preset.Pulses := 402_167_584;
   Par.Enc.Preset.Units := 348.56;
   Par.Enc.Config.Resolution := -125.663706143592;
   Par.Ax_Aut.SemiAut_Vel := 50.0;
   Par.Ax_Aut.Aut_Vel := 50.0;
   Par.Ax_Aut.Aut_Acc := 1.0;
   Par.Ax_Aut.Aut_Dec := 1.0;
   Par.Bloccaggio_Sens."2111B1".Enable := TRUE;
   Par.Bloccaggio_Sens."2111B1".RangeLow := 0.0;
   Par.Bloccaggio_Sens."2111B1".RangeHigh := 0.0;
END_DATA_BLOCK

DATA_BLOCK "A0302_Manipolatore_PERS"   // DB91
// stored: MemoryReserve 100
   VAR RETAIN
      Par : Struct
         Ax : "Positioning_EPOS_Machine_Par";
         Ax_Aut { S7_SetPoint := 'True'} : "A0301_Mach_Speed_Par";
         Ax_Pos : Struct
            Prelievo { S7_SetPoint := 'True'} : LReal := 0.0;
            BancoCtrl { S7_SetPoint := 'True'} : LReal := -648.0;
            BancoA0303 { S7_SetPoint := 'True'} : LReal := 545.0;
            Tollerance : Struct
               Prelievo { S7_SetPoint := 'True'} : LReal := 1.0;
               BancoCtrl { S7_SetPoint := 'True'} : LReal := 1.0;
               BancoA0303 { S7_SetPoint := 'True'} : LReal := 1.0;
            END_STRUCT;
         END_STRUCT;
      END_STRUCT;
      Pers_Data : Struct
         EncoderAbsolute_Preset_OK : Bool := TRUE;
         Persistent_ActualPosition : LReal := 0.0;
      END_STRUCT;
   END_VAR
BEGIN
   Par.Ax.PosTolerance := 0.5;
   Par.Ax.DelayInPosition := T#500MS;
   Par.Ax.Man_Vel := 10000.0;
   Par.Ax.Man_Acc := 1500.0;
   Par.Ax.Man_Dec := 1500.0;
   Par.Ax_Aut.SemiAut_Vel := 30000.0;
   Par.Ax_Aut.Aut_Vel := 30000.0;
   Par.Ax_Aut.Aut_Acc := 2000.0;
   Par.Ax_Aut.Aut_Dec := 2000.0;
END_DATA_BLOCK

DATA_BLOCK "Area0301_V_Counter"   // DB104
// stored: MemoryReserve 100
   VAR
      Value : LReal;
   END_VAR
BEGIN
END_DATA_BLOCK

DATA_BLOCK "A0302_Bordatrice_RegolazioneFormato_PERS"   // DB71
// stored: MemoryReserve 100
   VAR RETAIN
      Par_Machine : Struct
         Nervatura_Pos_Riposo : Real := 2.0;
         Passaggio01_MaxDisallineamentoAXs : Real := 0.5;   // (Controllo disabilitato se <= 0)
         Passaggio02_MaxDisallineamentoAXs : Real := 0.5;   // (Controllo disabilitato se <= 0)
         Passaggio03_MaxDisallineamentoAXs : Real := 0.5;   // (Controllo disabilitato se <= 0)
         Passaggio04_MaxDisallineamentoAXs : Real := 0.5;   // (Controllo disabilitato se <= 0)
         AxD_AutoSpeed { ExternalAccessible := 'False'; ExternalVisible := 'False'; ExternalWritable := 'False'} : Real := 100.0;
      END_STRUCT;
      Par_Enc : Array[1..9] of "PosFbk_RTN";
      Par_D { S7_SetPoint := 'True'} : Array[1..1] of "Positioning_DOL_Machine_Par";
      Par_M : Array[2..9] of "Positioning_MOL_Machine_Par";
      Pers_D { S7_SetPoint := 'True'} : Array[1..1] of "Positioning_DOL_Machine_Pers_Data";
      Pers_M : Array[2..9] of "Positioning_MOL_Machine_Pers_Data";
   END_VAR
BEGIN
   Par_Enc[1].Preset.Pulses := -1_814_114_496;
   Par_Enc[2].Preset.Pulses := -2_062_495_152;
   Par_Enc[3].Preset.Pulses := -1_142_247_532;
   Par_Enc[4].Preset.Pulses := 1_928_214_608;
   Par_Enc[5].Preset.Pulses := -519_364_864;
   Par_Enc[6].Preset.Pulses := -1_662_099_024;
   Par_Enc[7].Preset.Pulses := -1_564_817_400;
   Par_Enc[8].Preset.Pulses := 754_806_652;
   Par_Enc[9].Preset.Pulses := 904_129_836;
   Par_Enc[1].Preset.Units := 180.0;
   Par_Enc[2..9].Preset.Units := 45.0;
   Par_Enc[1].Config.Resolution := -0.2;
   Par_Enc[2..9].Config.Resolution := -1.0;
   Par_D[1].PosTolerance := 0.1;
   Par_D[1].Minus_Limit := 59.0;
   Par_D[1].Plus_Limit := 215.0;
   Par_D[1].PreCutOff := 0.1;
   Par_D[1].PreEndLowSpeed := 1.0;
   Par_D[1].PreEndMedSpeed := 5.0;
   Par_D[1].LowSpeed := 35.0;
   Par_D[1].MedSpeed := 70.0;
   Par_D[1].HighSpeed := 70.0;
   Par_D[1].Man_Speed := 100.0;
   Par_M[2..9].PosTolerance := 0.1;
   Par_M[2..9].DelayInPosition := T#100MS;
   Par_M[2..8].Minus_Limit := 38.0;
   Par_M[9].Minus_Limit := 38.5;
   Par_M[2..9].Plus_Limit := 52.0;
   Par_M[2..9].PreCutOff := 0.03;
   Pers_D[1].AxisHomed := TRUE;
   Pers_M[2..9].AxisHomed := TRUE;
END_DATA_BLOCK

DATA_BLOCK "A0302_OB30_Status"   // DB116
// stored: MemoryReserve 100
   VAR
      RETVAL_SET_CINT_Low : Int;
      RETVAL_SET_CINT_High : Int;
      RETVAL_QRY_CINT_Low : Int;
      RETVAL_QRY_CINT_High : Int;
      QRT_OB30_Low_CYCLE : UDInt;
      QRT_OB30_Low_PHASE : UDInt;
      QRT_OB30_Low_STATUS : Word;
      QRT_OB30_High_CYCLE : UDInt;
      QRT_OB30_High_PHASE : UDInt;
      QRT_OB30_High_STATUS : Word;
      OB30_Low : Bool;
      OB30_High : Bool;
   END_VAR
BEGIN
END_DATA_BLOCK

DATA_BLOCK "A0302_Bordatrice_PERS"   // DB44
// stored: MemoryReserve 100
   VAR RETAIN
      Par : Struct
         Ax_Man : "Positioning_EPOS_Machine_Par";
         Ax_Aut : "A0301_Mach_Speed_Par";
      END_STRUCT;
      Pers_Data : Struct
         EncoderAbsolute_Preset_OK : Bool := TRUE;
         Persistent_ActualPosition : LReal := 457025.036;
      END_STRUCT;
   END_VAR
BEGIN
   Par.Ax_Man.PosTolerance := 1.0;
   Par.Ax_Man.DelayInPosition := T#10MS;
   Par.Ax_Man.Man_Vel := 30000.0;
   Par.Ax_Man.Man_Acc := 1000.0;
   Par.Ax_Man.Man_Dec := 1000.0;
   Par.Ax_Aut.SemiAut_Vel := 40000.0;
   Par.Ax_Aut.Aut_Vel := 48000.0;
   Par.Ax_Aut.Aut_Acc := 1000.0;
   Par.Ax_Aut.Aut_Dec := 1000.0;
END_DATA_BLOCK

DATA_BLOCK "A0302_Rulliera_PERS"   // DB119
// stored: MemoryReserve 100
   VAR RETAIN
      Par : Struct
         Ax { S7_SetPoint := 'True'} : "SpeedMachine_Par";
         Ax_Aut { S7_SetPoint := 'True'} : "A0301_Mach_Speed_Par";
      END_STRUCT;
      IEC_SP : Struct
         FTC_CodaRall : Struct
            TON_PT : Time := T#300MS;
            TOF_PT : Time := T#300MS;
         END_STRUCT;
         FTC_CodaProxIng : Struct
            TON_PT : Time := T#300MS;
            TOF_PT : Time := T#300MS;
         END_STRUCT;
         FTC_Centro : Struct
            TON_PT : Time := T#300MS;
            TOF_PT : Time := T#300MS;
         END_STRUCT;
      END_STRUCT;
   END_VAR
BEGIN
   Par.Ax.Man.VelBwd := 2000.0;
   Par.Ax.Man.VelFwdHigh := 50000.0;
   Par.Ax.Man.VelFwdLow := 20000.0;
   Par.Ax.Man.Acc := 2000.0;
   Par.Ax.Man.Dec := 2000.0;
   Par.Ax.Man.DelayChangeVel := T#200MS;
   Par.Ax_Aut.SemiAut_Vel := 35000.0;
   Par.Ax_Aut.Aut_Vel := 30000.0;
   Par.Ax_Aut.Aut_Acc := 1100.0;
   Par.Ax_Aut.Aut_Dec := 1100.0;
END_DATA_BLOCK

ORGANIZATION_BLOCK "A03_OB1"   // OB1, LAD, ProgramCycle
TITLE = "Main Program Sweep (Cycle)"
// stored: SetENOAutomatically false
   VAR_INPUT
      Initial_Call : Bool;   // Initial call of this OB
      Remanence : Bool;   // =True, if remanent data are available
   END_VAR
BEGIN

REGION Network 1
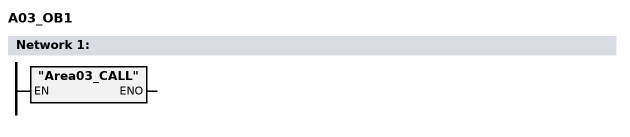
   RUNG wire#powerrail
      "Area03_CALL"()
   END_RUNG
   // the same network as SCL:
   "Area03_CALL"();
END_REGION
END_ORGANIZATION_BLOCK

FUNCTION "Area03_CALL" : Void   // FC61, LAD
TITLE = Area 03
// stored: SetENOAutomatically false
   VAR_TEMP
      AlrIndex : Int;
      WngIndex : Int;
      MissingOutput : Bool;
   END_VAR
BEGIN

REGION Network 1: Data In
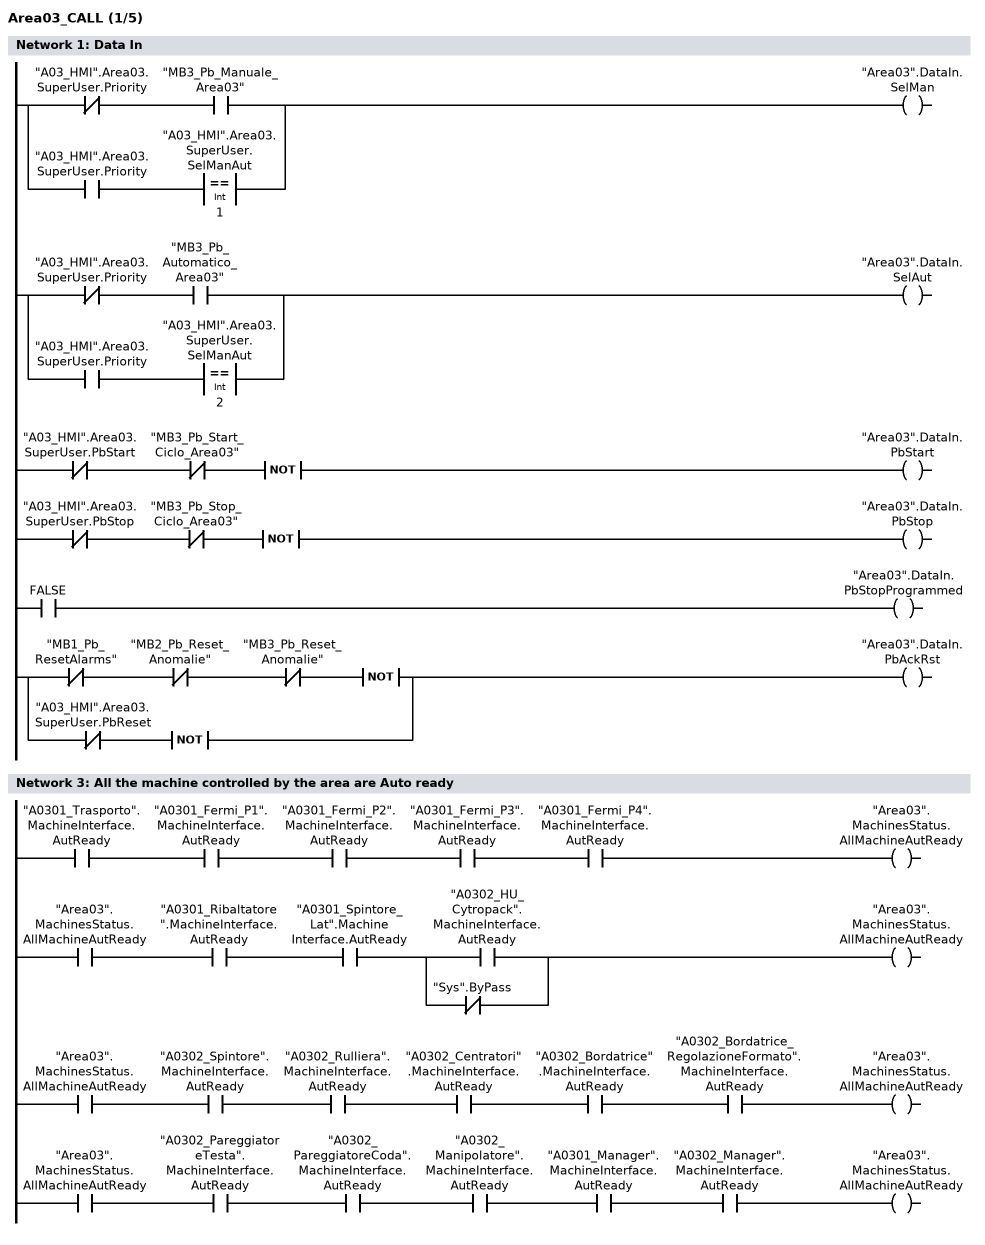
   RUNG wire#powerrail
      I_Contact( "A03_HMI".Area03.SuperUser.Priority )
      Contact( "MB3_Pb_Manuale_Area03" )
      wire#w1
      Coil( "Area03".DataIn.SelMan )
   END_RUNG
   RUNG wire#powerrail
      Contact( "A03_HMI".Area03.SuperUser.Priority )
      { S7_Templates := "SrcType := Int" } EQ_Contact(in1 := "A03_HMI".Area03.SuperUser.SelManAut, in2 := 1)
   END_RUNG wire#w1
   RUNG wire#powerrail
      I_Contact( "A03_HMI".Area03.SuperUser.Priority )
      Contact( "MB3_Pb_Automatico_Area03" )
      wire#w2
      Coil( "Area03".DataIn.SelAut )
   END_RUNG
   RUNG wire#powerrail
      Contact( "A03_HMI".Area03.SuperUser.Priority )
      { S7_Templates := "SrcType := Int" } EQ_Contact(in1 := "A03_HMI".Area03.SuperUser.SelManAut, in2 := 2)
   END_RUNG wire#w2
   RUNG wire#powerrail
      I_Contact( "A03_HMI".Area03.SuperUser.PbStart )
      I_Contact( "MB3_Pb_Start_Ciclo_Area03" )
      Not()
      Coil( "Area03".DataIn.PbStart )
   END_RUNG
   RUNG wire#powerrail
      I_Contact( "A03_HMI".Area03.SuperUser.PbStop )
      I_Contact( "MB3_Pb_Stop_Ciclo_Area03" )
      Not()
      Coil( "Area03".DataIn.PbStop )
   END_RUNG
   RUNG wire#powerrail
      Contact( FALSE )
      Coil( "Area03".DataIn.PbStopProgrammed )
   END_RUNG
   RUNG wire#powerrail
      I_Contact( "MB1_Pb_ResetAlarms" )
      I_Contact( "MB2_Pb_Reset_Anomalie" )
      I_Contact( "MB3_Pb_Reset_Anomalie" )
      Not()
      wire#w3
      Coil( "Area03".DataIn.PbAckRst )
   END_RUNG
   RUNG wire#powerrail
      I_Contact( "A03_HMI".Area03.SuperUser.PbReset )
      Not()
   END_RUNG wire#w3
   // the same network as SCL:
   "Area03".DataIn.SelMan := (NOT "A03_HMI".Area03.SuperUser.Priority AND "MB3_Pb_Manuale_Area03") OR ("A03_HMI".Area03.SuperUser.Priority AND ("A03_HMI".Area03.SuperUser.SelManAut = 1));
   "Area03".DataIn.SelAut := (NOT "A03_HMI".Area03.SuperUser.Priority AND "MB3_Pb_Automatico_Area03") OR ("A03_HMI".Area03.SuperUser.Priority AND ("A03_HMI".Area03.SuperUser.SelManAut = 2));
   "Area03".DataIn.PbStart := NOT (NOT "A03_HMI".Area03.SuperUser.PbStart AND NOT "MB3_Pb_Start_Ciclo_Area03");
   "Area03".DataIn.PbStop := NOT (NOT "A03_HMI".Area03.SuperUser.PbStop AND NOT "MB3_Pb_Stop_Ciclo_Area03");
   "Area03".DataIn.PbStopProgrammed := FALSE;
   "Area03".DataIn.PbAckRst := NOT (NOT "MB1_Pb_ResetAlarms" AND NOT "MB2_Pb_Reset_Anomalie" AND NOT "MB3_Pb_Reset_Anomalie") OR NOT (NOT "A03_HMI".Area03.SuperUser.PbReset);
END_REGION

REGION Network 3: All the machine controlled by the area are Auto ready
   RUNG wire#powerrail
      Contact( "A0301_Trasporto".MachineInterface.AutReady )
      Contact( "A0301_Fermi_P1".MachineInterface.AutReady )
      Contact( "A0301_Fermi_P2".MachineInterface.AutReady )
      Contact( "A0301_Fermi_P3".MachineInterface.AutReady )
      Contact( "A0301_Fermi_P4".MachineInterface.AutReady )
      Coil( "Area03".MachinesStatus.AllMachineAutReady )
   END_RUNG
   RUNG wire#powerrail
      Contact( "Area03".MachinesStatus.AllMachineAutReady )
      Contact( "A0301_Ribaltatore".MachineInterface.AutReady )
      Contact( "A0301_Spintore_Lat".MachineInterface.AutReady )
      wire#w1
      Contact( "A0302_HU_Cytropack".MachineInterface.AutReady )
      wire#w2
      Coil( "Area03".MachinesStatus.AllMachineAutReady )
   END_RUNG
   RUNG wire#w1
      I_Contact( "Sys".ByPass )
   END_RUNG wire#w2
   RUNG wire#powerrail
      Contact( "Area03".MachinesStatus.AllMachineAutReady )
      Contact( "A0302_Spintore".MachineInterface.AutReady )
      Contact( "A0302_Rulliera".MachineInterface.AutReady )
      Contact( "A0302_Centratori".MachineInterface.AutReady )
      Contact( "A0302_Bordatrice".MachineInterface.AutReady )
      Contact( "A0302_Bordatrice_RegolazioneFormato".MachineInterface.AutReady )
      Coil( "Area03".MachinesStatus.AllMachineAutReady )
   END_RUNG
   RUNG wire#powerrail
      Contact( "Area03".MachinesStatus.AllMachineAutReady )
      Contact( "A0302_PareggiatoreTesta".MachineInterface.AutReady )
      Contact( "A0302_PareggiatoreCoda".MachineInterface.AutReady )
      Contact( "A0302_Manipolatore".MachineInterface.AutReady )
      Contact( "A0301_Manager".MachineInterface.AutReady )
      Contact( "A0302_Manager".MachineInterface.AutReady )
      Coil( "Area03".MachinesStatus.AllMachineAutReady )
   END_RUNG
   // the same network as SCL:
   "Area03".MachinesStatus.AllMachineAutReady := "A0301_Trasporto".MachineInterface.AutReady AND "A0301_Fermi_P1".MachineInterface.AutReady AND "A0301_Fermi_P2".MachineInterface.AutReady AND "A0301_Fermi_P3".MachineInterface.AutReady AND "A0301_Fermi_P4".MachineInterface.AutReady;
   "Area03".MachinesStatus.AllMachineAutReady := "Area03".MachinesStatus.AllMachineAutReady AND "A0301_Ribaltatore".MachineInterface.AutReady AND "A0301_Spintore_Lat".MachineInterface.AutReady AND ("A0302_HU_Cytropack".MachineInterface.AutReady OR NOT "Sys".ByPass);
   "Area03".MachinesStatus.AllMachineAutReady := "Area03".MachinesStatus.AllMachineAutReady AND "A0302_Spintore".MachineInterface.AutReady AND "A0302_Rulliera".MachineInterface.AutReady AND "A0302_Centratori".MachineInterface.AutReady AND "A0302_Bordatrice".MachineInterface.AutReady AND "A0302_Bordatrice_RegolazioneFormato".MachineInterface.AutReady;
   "Area03".MachinesStatus.AllMachineAutReady := "Area03".MachinesStatus.AllMachineAutReady AND "A0302_PareggiatoreTesta".MachineInterface.AutReady AND "A0302_PareggiatoreCoda".MachineInterface.AutReady AND "A0302_Manipolatore".MachineInterface.AutReady AND "A0301_Manager".MachineInterface.AutReady AND "A0302_Manager".MachineInterface.AutReady;
END_REGION

REGION Network 4: One of machine controlled by the area is aborting
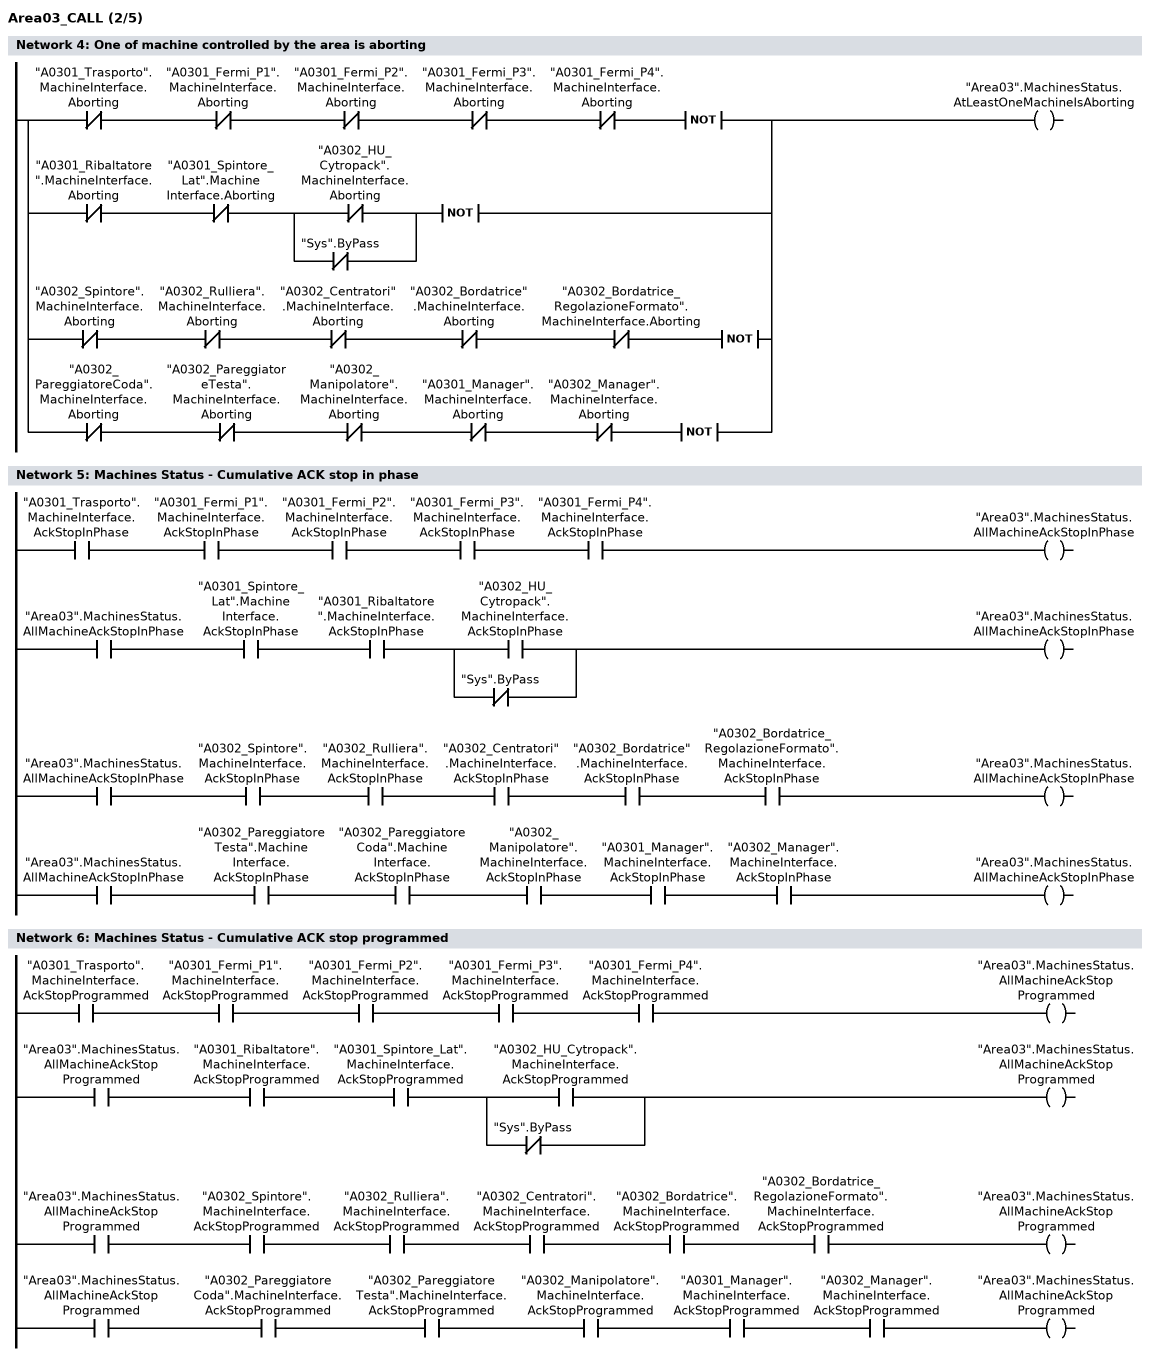
   RUNG wire#powerrail
      I_Contact( "A0301_Trasporto".MachineInterface.Aborting )
      I_Contact( "A0301_Fermi_P1".MachineInterface.Aborting )
      I_Contact( "A0301_Fermi_P2".MachineInterface.Aborting )
      I_Contact( "A0301_Fermi_P3".MachineInterface.Aborting )
      I_Contact( "A0301_Fermi_P4".MachineInterface.Aborting )
      Not()
      wire#w1
      Coil( "Area03".MachinesStatus.AtLeastOneMachineIsAborting )
   END_RUNG
   RUNG wire#powerrail
      I_Contact( "A0301_Ribaltatore".MachineInterface.Aborting )
      I_Contact( "A0301_Spintore_Lat".MachineInterface.Aborting )
      wire#w2
      I_Contact( "A0302_HU_Cytropack".MachineInterface.Aborting )
      wire#w3
      Not()
   END_RUNG wire#w1
   RUNG wire#w2
      I_Contact( "Sys".ByPass )
   END_RUNG wire#w3
   RUNG wire#powerrail
      I_Contact( "A0302_Spintore".MachineInterface.Aborting )
      I_Contact( "A0302_Rulliera".MachineInterface.Aborting )
      I_Contact( "A0302_Centratori".MachineInterface.Aborting )
      I_Contact( "A0302_Bordatrice".MachineInterface.Aborting )
      I_Contact( "A0302_Bordatrice_RegolazioneFormato".MachineInterface.Aborting )
      Not()
   END_RUNG wire#w1
   RUNG wire#powerrail
      I_Contact( "A0302_PareggiatoreCoda".MachineInterface.Aborting )
      I_Contact( "A0302_PareggiatoreTesta".MachineInterface.Aborting )
      I_Contact( "A0302_Manipolatore".MachineInterface.Aborting )
      I_Contact( "A0301_Manager".MachineInterface.Aborting )
      I_Contact( "A0302_Manager".MachineInterface.Aborting )
      Not()
   END_RUNG wire#w1
   // the same network as SCL:
   "Area03".MachinesStatus.AtLeastOneMachineIsAborting := NOT (NOT "A0301_Trasporto".MachineInterface.Aborting AND NOT "A0301_Fermi_P1".MachineInterface.Aborting AND NOT "A0301_Fermi_P2".MachineInterface.Aborting AND NOT "A0301_Fermi_P3".MachineInterface.Aborting AND NOT "A0301_Fermi_P4".MachineInterface.Aborting) OR NOT (NOT "A0301_Ribaltatore".MachineInterface.Aborting AND NOT "A0301_Spintore_Lat".MachineInterface.Aborting AND (NOT "A0302_HU_Cytropack".MachineInterface.Aborting OR NOT "Sys".ByPass)) OR NOT (NOT "A0302_Spintore".MachineInterface.Aborting AND NOT "A0302_Rulliera".MachineInterface.Aborting AND NOT "A0302_Centratori".MachineInterface.Aborting AND NOT "A0302_Bordatrice".MachineInterface.Aborting AND NOT "A0302_Bordatrice_RegolazioneFormato".MachineInterface.Aborting) OR NOT (NOT "A0302_PareggiatoreCoda".MachineInterface.Aborting AND NOT "A0302_PareggiatoreTesta".MachineInterface.Aborting AND NOT "A0302_Manipolatore".MachineInterface.Aborting AND NOT "A0301_Manager".MachineInterface.Aborting AND NOT "A0302_Manager".MachineInterface.Aborting);
END_REGION

REGION Network 5: Machines Status - Cumulative ACK stop in phase
   RUNG wire#powerrail
      Contact( "A0301_Trasporto".MachineInterface.AckStopInPhase )
      Contact( "A0301_Fermi_P1".MachineInterface.AckStopInPhase )
      Contact( "A0301_Fermi_P2".MachineInterface.AckStopInPhase )
      Contact( "A0301_Fermi_P3".MachineInterface.AckStopInPhase )
      Contact( "A0301_Fermi_P4".MachineInterface.AckStopInPhase )
      Coil( "Area03".MachinesStatus.AllMachineAckStopInPhase )
   END_RUNG
   RUNG wire#powerrail
      Contact( "Area03".MachinesStatus.AllMachineAckStopInPhase )
      Contact( "A0301_Spintore_Lat".MachineInterface.AckStopInPhase )
      Contact( "A0301_Ribaltatore".MachineInterface.AckStopInPhase )
      wire#w1
      Contact( "A0302_HU_Cytropack".MachineInterface.AckStopInPhase )
      wire#w2
      Coil( "Area03".MachinesStatus.AllMachineAckStopInPhase )
   END_RUNG
   RUNG wire#w1
      I_Contact( "Sys".ByPass )
   END_RUNG wire#w2
   RUNG wire#powerrail
      Contact( "Area03".MachinesStatus.AllMachineAckStopInPhase )
      Contact( "A0302_Spintore".MachineInterface.AckStopInPhase )
      Contact( "A0302_Rulliera".MachineInterface.AckStopInPhase )
      Contact( "A0302_Centratori".MachineInterface.AckStopInPhase )
      Contact( "A0302_Bordatrice".MachineInterface.AckStopInPhase )
      Contact( "A0302_Bordatrice_RegolazioneFormato".MachineInterface.AckStopInPhase )
      Coil( "Area03".MachinesStatus.AllMachineAckStopInPhase )
   END_RUNG
   RUNG wire#powerrail
      Contact( "Area03".MachinesStatus.AllMachineAckStopInPhase )
      Contact( "A0302_PareggiatoreTesta".MachineInterface.AckStopInPhase )
      Contact( "A0302_PareggiatoreCoda".MachineInterface.AckStopInPhase )
      Contact( "A0302_Manipolatore".MachineInterface.AckStopInPhase )
      Contact( "A0301_Manager".MachineInterface.AckStopInPhase )
      Contact( "A0302_Manager".MachineInterface.AckStopInPhase )
      Coil( "Area03".MachinesStatus.AllMachineAckStopInPhase )
   END_RUNG
   // the same network as SCL:
   "Area03".MachinesStatus.AllMachineAckStopInPhase := "A0301_Trasporto".MachineInterface.AckStopInPhase AND "A0301_Fermi_P1".MachineInterface.AckStopInPhase AND "A0301_Fermi_P2".MachineInterface.AckStopInPhase AND "A0301_Fermi_P3".MachineInterface.AckStopInPhase AND "A0301_Fermi_P4".MachineInterface.AckStopInPhase;
   "Area03".MachinesStatus.AllMachineAckStopInPhase := "Area03".MachinesStatus.AllMachineAckStopInPhase AND "A0301_Spintore_Lat".MachineInterface.AckStopInPhase AND "A0301_Ribaltatore".MachineInterface.AckStopInPhase AND ("A0302_HU_Cytropack".MachineInterface.AckStopInPhase OR NOT "Sys".ByPass);
   "Area03".MachinesStatus.AllMachineAckStopInPhase := "Area03".MachinesStatus.AllMachineAckStopInPhase AND "A0302_Spintore".MachineInterface.AckStopInPhase AND "A0302_Rulliera".MachineInterface.AckStopInPhase AND "A0302_Centratori".MachineInterface.AckStopInPhase AND "A0302_Bordatrice".MachineInterface.AckStopInPhase AND "A0302_Bordatrice_RegolazioneFormato".MachineInterface.AckStopInPhase;
   "Area03".MachinesStatus.AllMachineAckStopInPhase := "Area03".MachinesStatus.AllMachineAckStopInPhase AND "A0302_PareggiatoreTesta".MachineInterface.AckStopInPhase AND "A0302_PareggiatoreCoda".MachineInterface.AckStopInPhase AND "A0302_Manipolatore".MachineInterface.AckStopInPhase AND "A0301_Manager".MachineInterface.AckStopInPhase AND "A0302_Manager".MachineInterface.AckStopInPhase;
END_REGION

REGION Network 6: Machines Status - Cumulative ACK stop programmed
   RUNG wire#powerrail
      Contact( "A0301_Trasporto".MachineInterface.AckStopProgrammed )
      Contact( "A0301_Fermi_P1".MachineInterface.AckStopProgrammed )
      Contact( "A0301_Fermi_P2".MachineInterface.AckStopProgrammed )
      Contact( "A0301_Fermi_P3".MachineInterface.AckStopProgrammed )
      Contact( "A0301_Fermi_P4".MachineInterface.AckStopProgrammed )
      Coil( "Area03".MachinesStatus.AllMachineAckStopProgrammed )
   END_RUNG
   RUNG wire#powerrail
      Contact( "Area03".MachinesStatus.AllMachineAckStopProgrammed )
      Contact( "A0301_Ribaltatore".MachineInterface.AckStopProgrammed )
      Contact( "A0301_Spintore_Lat".MachineInterface.AckStopProgrammed )
      wire#w1
      Contact( "A0302_HU_Cytropack".MachineInterface.AckStopProgrammed )
      wire#w2
      Coil( "Area03".MachinesStatus.AllMachineAckStopProgrammed )
   END_RUNG
   RUNG wire#w1
      I_Contact( "Sys".ByPass )
   END_RUNG wire#w2
   RUNG wire#powerrail
      Contact( "Area03".MachinesStatus.AllMachineAckStopProgrammed )
      Contact( "A0302_Spintore".MachineInterface.AckStopProgrammed )
      Contact( "A0302_Rulliera".MachineInterface.AckStopProgrammed )
      Contact( "A0302_Centratori".MachineInterface.AckStopProgrammed )
      Contact( "A0302_Bordatrice".MachineInterface.AckStopProgrammed )
      Contact( "A0302_Bordatrice_RegolazioneFormato".MachineInterface.AckStopProgrammed )
      Coil( "Area03".MachinesStatus.AllMachineAckStopProgrammed )
   END_RUNG
   RUNG wire#powerrail
      Contact( "Area03".MachinesStatus.AllMachineAckStopProgrammed )
      Contact( "A0302_PareggiatoreCoda".MachineInterface.AckStopProgrammed )
      Contact( "A0302_PareggiatoreTesta".MachineInterface.AckStopProgrammed )
      Contact( "A0302_Manipolatore".MachineInterface.AckStopProgrammed )
      Contact( "A0301_Manager".MachineInterface.AckStopProgrammed )
      Contact( "A0302_Manager".MachineInterface.AckStopProgrammed )
      Coil( "Area03".MachinesStatus.AllMachineAckStopProgrammed )
   END_RUNG
   // the same network as SCL:
   "Area03".MachinesStatus.AllMachineAckStopProgrammed := "A0301_Trasporto".MachineInterface.AckStopProgrammed AND "A0301_Fermi_P1".MachineInterface.AckStopProgrammed AND "A0301_Fermi_P2".MachineInterface.AckStopProgrammed AND "A0301_Fermi_P3".MachineInterface.AckStopProgrammed AND "A0301_Fermi_P4".MachineInterface.AckStopProgrammed;
   "Area03".MachinesStatus.AllMachineAckStopProgrammed := "Area03".MachinesStatus.AllMachineAckStopProgrammed AND "A0301_Ribaltatore".MachineInterface.AckStopProgrammed AND "A0301_Spintore_Lat".MachineInterface.AckStopProgrammed AND ("A0302_HU_Cytropack".MachineInterface.AckStopProgrammed OR NOT "Sys".ByPass);
   "Area03".MachinesStatus.AllMachineAckStopProgrammed := "Area03".MachinesStatus.AllMachineAckStopProgrammed AND "A0302_Spintore".MachineInterface.AckStopProgrammed AND "A0302_Rulliera".MachineInterface.AckStopProgrammed AND "A0302_Centratori".MachineInterface.AckStopProgrammed AND "A0302_Bordatrice".MachineInterface.AckStopProgrammed AND "A0302_Bordatrice_RegolazioneFormato".MachineInterface.AckStopProgrammed;
   "Area03".MachinesStatus.AllMachineAckStopProgrammed := "Area03".MachinesStatus.AllMachineAckStopProgrammed AND "A0302_PareggiatoreCoda".MachineInterface.AckStopProgrammed AND "A0302_PareggiatoreTesta".MachineInterface.AckStopProgrammed AND "A0302_Manipolatore".MachineInterface.AckStopProgrammed AND "A0301_Manager".MachineInterface.AckStopProgrammed AND "A0302_Manager".MachineInterface.AckStopProgrammed;
END_REGION

